Yaskawa INFORM job: new_kufsa_updated.JBI

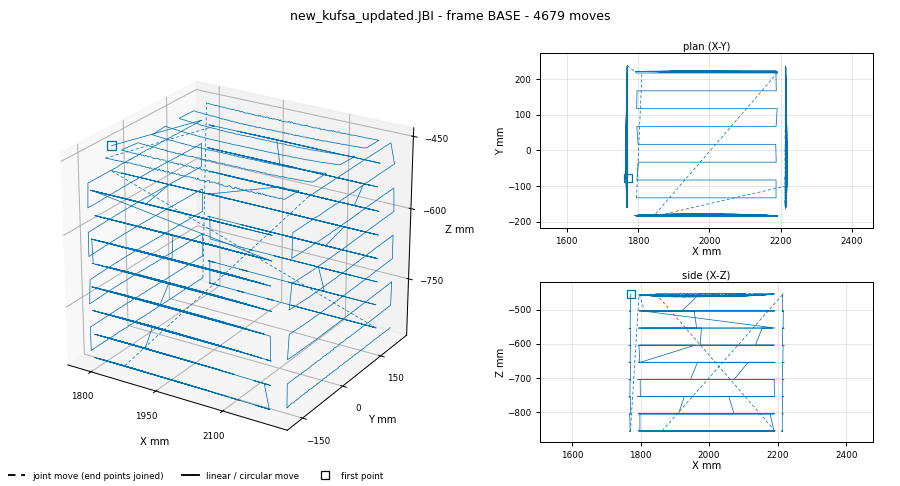
[picture p0: tool path of new_kufsa_updated.JBI in frame BASE, 4679 of 4679 moves have a stored position in this frame; points joined in program order, loops and branches not executed]
/JOB
//NAME NEW_KUFSA
//POS
///NPOS 4679,0,0,0,0,0
///TOOL 0
///POSTYPE BASE
///RECTAN
///RCONF 1,0,0,0,0,0,0,0,0,0,0,0,0,0,0,0,0,0,0,0,0,0,0,0
C00000=1771.695900,-78.143700,-454.553300,-91.472712,-88.665219,-178.527919
C00001=1770.552300,237.577800,-504.553300,-91.472712,-88.665219,-178.527919
C00002=1770.327900,234.301700,-504.553300,-91.472712,-88.665219,-178.527919
C00003=1770.357500,229.959000,-504.553300,-91.472712,-88.665219,-178.527919
C00004=1770.715100,226.685000,-504.553300,-91.472712,-88.665219,-178.527919
C00005=1770.694700,222.913600,-504.553300,-91.472712,-88.665219,-178.527919
C00006=1770.618200,221.900700,-504.553300,-91.472712,-88.665219,-178.527919
C00007=1770.622400,218.998600,-504.553300,-91.472712,-88.665219,-178.527919
C00008=1770.451600,217.707000,-504.553300,-91.472712,-88.665219,-178.527919
C00009=1770.752700,214.366400,-504.553300,-91.472712,-88.665219,-178.527919
C00010=1770.697000,210.035600,-504.553300,-91.472712,-88.665219,-178.527919
C00011=1770.753100,207.951700,-504.553300,-91.472712,-88.665219,-178.527919
C00012=1770.680200,203.374600,-504.553300,-91.472712,-88.665219,-178.527919
C00013=1770.529700,199.363700,-504.553300,-91.472712,-88.665219,-178.527919
C00014=1770.704300,193.088900,-504.553300,-91.472712,-88.665219,-178.527919
C00015=1770.481900,189.234700,-504.553300,-91.472712,-88.665219,-178.527919
C00016=1770.674300,186.293400,-504.553300,-91.472712,-88.665219,-178.527919
C00017=1770.533500,181.144000,-504.553300,-91.472712,-88.665219,-178.527919
C00018=1770.619900,177.321600,-504.553300,-91.472712,-88.665219,-178.527919
C00019=1770.311100,172.891400,-504.553300,-91.472712,-88.665219,-178.527919
C00020=1770.213900,166.678800,-504.553300,-91.472712,-88.665219,-178.527919
C00021=1770.097800,164.479000,-504.553300,-91.472712,-88.665219,-178.527919
C00022=1769.937500,159.949500,-504.553300,-91.472712,-88.665219,-178.527919
C00023=1770.653000,157.893100,-504.553300,-91.472712,-88.665219,-178.527919
C00024=1770.749700,154.381500,-504.553300,-91.472712,-88.665219,-178.527919
C00025=1770.288500,151.107400,-504.553300,-91.472712,-88.665219,-178.527919
C00026=1770.668700,148.632000,-504.553300,-91.472712,-88.665219,-178.527919
C00027=1770.398300,145.757600,-504.553300,-91.472712,-88.665219,-178.527919
C00028=1769.498100,142.997800,-504.553300,-91.472712,-88.665219,-178.527919
C00029=1769.363100,139.160700,-504.553300,-91.472712,-88.665219,-178.527919
C00030=1769.459100,135.555500,-504.553300,-91.472712,-88.665219,-178.527919
C00031=1769.040900,132.650400,-504.553300,-91.472712,-88.665219,-178.527919
C00032=1769.898800,130.507300,-504.553300,-91.472712,-88.665219,-178.527919
C00033=1770.728700,127.335900,-504.553300,-91.472712,-88.665219,-178.527919
C00034=1770.427200,123.559800,-504.553300,-91.472712,-88.665219,-178.527919
C00035=1768.954900,119.644000,-504.553300,-91.472712,-88.665219,-178.527919
C00036=1769.993600,117.378600,-504.553300,-91.472712,-88.665219,-178.527919
C00037=1768.828100,114.262100,-504.553300,-91.472712,-88.665219,-178.527919
C00038=1770.115200,111.383800,-504.553300,-91.472712,-88.665219,-178.527919
C00039=1769.668100,108.550000,-504.553300,-91.472712,-88.665219,-178.527919
C00040=1768.761100,104.884700,-504.553300,-91.472712,-88.665219,-178.527919
C00041=1769.568000,102.393100,-504.553300,-91.472712,-88.665219,-178.527919
C00042=1770.193300,98.407500,-504.553300,-91.472712,-88.665219,-178.527919
C00043=1768.903700,96.183100,-504.553300,-91.472712,-88.665219,-178.527919
C00044=1768.807500,91.494800,-504.553300,-91.472712,-88.665219,-178.527919
C00045=1769.610500,88.437300,-504.553300,-91.472712,-88.665219,-178.527919
C00046=1769.643300,85.334200,-504.553300,-91.472712,-88.665219,-178.527919
C00047=1770.204500,83.163200,-504.553300,-91.472712,-88.665219,-178.527919
C00048=1769.143800,79.495600,-504.553300,-91.472712,-88.665219,-178.527919
C00049=1770.143500,76.022500,-504.553300,-91.472712,-88.665219,-178.527919
C00050=1770.166100,73.523800,-504.553300,-91.472712,-88.665219,-178.527919
C00051=1768.794300,69.839900,-504.553300,-91.472712,-88.665219,-178.527919
C00052=1768.256500,65.364800,-504.553300,-91.472712,-88.665219,-178.527919
C00053=1769.079700,62.108500,-504.553300,-91.472712,-88.665219,-178.527919
C00054=1769.961500,58.974300,-504.553300,-91.472712,-88.665219,-178.527919
C00055=1770.647500,53.217300,-504.553300,-91.472712,-88.665219,-178.527919
C00056=1769.116700,51.163800,-504.553300,-91.472712,-88.665219,-178.527919
C00057=1768.800500,45.123900,-504.553300,-91.472712,-88.665219,-178.527919
C00058=1768.002400,42.027000,-504.553300,-91.472712,-88.665219,-178.527919
C00059=1768.569100,38.028400,-504.553300,-91.472712,-88.665219,-178.527919
C00060=1769.872300,32.986500,-504.553300,-91.472712,-88.665219,-178.527919
C00061=1768.268600,29.407100,-504.553300,-91.472712,-88.665219,-178.527919
C00062=1768.741300,27.721600,-504.553300,-91.472712,-88.665219,-178.527919
C00063=1768.516100,24.486500,-504.553300,-91.472712,-88.665219,-178.527919
C00064=1768.709900,22.063000,-504.553300,-91.472712,-88.665219,-178.527919
C00065=1770.169000,18.529100,-504.553300,-91.472712,-88.665219,-178.527919
C00066=1769.338300,14.603500,-504.553300,-91.472712,-88.665219,-178.527919
C00067=1769.785200,12.781600,-504.553300,-91.472712,-88.665219,-178.527919
C00068=1768.917400,10.596100,-504.553300,-91.472712,-88.665219,-178.527919
C00069=1770.959800,8.457400,-504.553300,-91.472712,-88.665219,-178.527919
C00070=1770.078300,4.762700,-504.553300,-91.472712,-88.665219,-178.527919
C00071=1770.056300,0.334200,-504.553300,-91.472712,-88.665219,-178.527919
C00072=1768.340800,-1.831400,-504.553300,-91.472712,-88.665219,-178.527919
C00073=1770.254300,-5.058200,-504.553300,-91.472712,-88.665219,-178.527919
C00074=1769.677500,-8.070100,-504.553300,-91.472712,-88.665219,-178.527919
C00075=1770.879300,-10.712700,-504.553300,-91.472712,-88.665219,-178.527919
C00076=1768.750700,-14.573600,-504.553300,-91.472712,-88.665219,-178.527919
C00077=1770.340400,-15.957100,-504.553300,-91.472712,-88.665219,-178.527919
C00078=1768.733600,-20.306900,-504.553300,-91.472712,-88.665219,-178.527919
C00079=1769.800500,-22.681600,-504.553300,-91.472712,-88.665219,-178.527919
C00080=1769.413100,-26.458000,-504.553300,-91.472712,-88.665219,-178.527919
C00081=1769.645800,-30.948700,-504.553300,-91.472712,-88.665219,-178.527919
C00082=1769.732900,-34.377100,-504.553300,-91.472712,-88.665219,-178.527919
C00083=1769.999900,-36.989700,-504.553300,-91.472712,-88.665219,-178.527919
C00084=1768.941700,-40.940500,-504.553300,-91.472712,-88.665219,-178.527919
C00085=1769.293400,-44.109800,-504.553300,-91.472712,-88.665219,-178.527919
C00086=1769.076200,-46.979100,-504.553300,-91.472712,-88.665219,-178.527919
C00087=1769.685800,-51.575500,-504.553300,-91.472712,-88.665219,-178.527919
C00088=1769.818600,-53.702900,-504.553300,-91.472712,-88.665219,-178.527919
C00089=1771.044100,-58.594600,-504.553300,-91.472712,-88.665219,-178.527919
C00090=1770.444400,-61.359500,-504.553300,-91.472712,-88.665219,-178.527919
C00091=1771.083300,-65.467700,-504.553300,-91.472712,-88.665219,-178.527919
C00092=1770.718600,-67.730300,-504.553300,-91.472712,-88.665219,-178.527919
C00093=1770.401400,-71.308800,-504.553300,-91.472712,-88.665219,-178.527919
C00094=1770.970400,-75.459300,-504.553300,-91.472712,-88.665219,-178.527919
C00095=1770.670500,-79.143800,-504.553300,-91.472712,-88.665219,-178.527919
C00096=1769.980400,-82.193500,-504.553300,-91.472712,-88.665219,-178.527919
C00097=1771.083500,-85.926000,-504.553300,-91.472712,-88.665219,-178.527919
C00098=1770.271700,-88.724100,-504.553300,-91.472712,-88.665219,-178.527919
C00099=1770.893900,-91.597400,-504.553300,-91.472712,-88.665219,-178.527919
C00100=1770.927400,-97.401600,-504.553300,-91.472712,-88.665219,-178.527919
C00101=1770.186700,-101.527400,-504.553300,-91.472712,-88.665219,-178.527919
C00102=1771.038900,-105.643300,-504.553300,-91.472712,-88.665219,-178.527919
C00103=1770.472200,-109.502300,-504.553300,-91.472712,-88.665219,-178.527919
C00104=1771.164000,-113.253700,-504.553300,-91.472712,-88.665219,-178.527919
C00105=1770.459300,-119.489700,-504.553300,-91.472712,-88.665219,-178.527919
C00106=1770.831500,-123.480600,-504.553300,-91.472712,-88.665219,-178.527919
C00107=1770.300700,-127.391200,-504.553300,-91.472712,-88.665219,-178.527919
C00108=1770.407700,-131.896000,-504.553300,-91.472712,-88.665219,-178.527919
C00109=1770.835300,-137.199200,-504.553300,-91.472712,-88.665219,-178.527919
C00110=1770.659300,-142.340600,-504.553300,-91.472712,-88.665219,-178.527919
C00111=1770.414300,-146.357400,-504.553300,-91.472712,-88.665219,-178.527919
C00112=1770.891300,-148.126700,-504.553300,-91.472712,-88.665219,-178.527919
C00113=1770.958700,-151.548700,-504.553300,-91.472712,-88.665219,-178.527919
C00114=1770.369300,-155.780700,-504.553300,-91.472712,-88.665219,-178.527919
C00115=1770.064400,-157.972700,-554.553300,-91.472712,-88.665219,-178.527919
C00116=1769.985800,-154.798600,-554.553300,-91.472712,-88.665219,-178.527919
C00117=1770.252900,-151.668100,-554.553300,-91.472712,-88.665219,-178.527919
C00118=1770.186000,-148.149800,-554.553300,-91.472712,-88.665219,-178.527919
C00119=1769.926300,-145.462600,-554.553300,-91.472712,-88.665219,-178.527919
C00120=1770.034700,-142.677400,-554.553300,-91.472712,-88.665219,-178.527919
C00121=1770.051100,-141.018200,-554.553300,-91.472712,-88.665219,-178.527919
C00122=1770.290900,-137.062400,-554.553300,-91.472712,-88.665219,-178.527919
C00123=1770.018000,-133.335900,-554.553300,-91.472712,-88.665219,-178.527919
C00124=1769.803300,-128.424000,-554.553300,-91.472712,-88.665219,-178.527919
C00125=1769.855600,-124.269200,-554.553300,-91.472712,-88.665219,-178.527919
C00126=1769.525500,-118.390000,-554.553300,-91.472712,-88.665219,-178.527919
C00127=1769.793500,-115.424000,-554.553300,-91.472712,-88.665219,-178.527919
C00128=1769.519200,-110.220900,-554.553300,-91.472712,-88.665219,-178.527919
C00129=1769.684400,-107.152900,-554.553300,-91.472712,-88.665219,-178.527919
C00130=1768.914900,-102.406800,-554.553300,-91.472712,-88.665219,-178.527919
C00131=1769.115300,-98.536800,-554.553300,-91.472712,-88.665219,-178.527919
C00132=1769.053600,-93.635300,-554.553300,-91.472712,-88.665219,-178.527919
C00133=1769.429700,-91.018400,-554.553300,-91.472712,-88.665219,-178.527919
C00134=1768.813100,-86.595600,-554.553300,-91.472712,-88.665219,-178.527919
C00135=1768.570100,-84.367200,-554.553300,-91.472712,-88.665219,-178.527919
C00136=1768.957000,-77.814700,-554.553300,-91.472712,-88.665219,-178.527919
C00137=1768.595600,-74.979800,-554.553300,-91.472712,-88.665219,-178.527919
C00138=1768.799500,-71.746300,-554.553300,-91.472712,-88.665219,-178.527919
C00139=1768.054600,-65.699200,-554.553300,-91.472712,-88.665219,-178.527919
C00140=1768.662200,-62.089600,-554.553300,-91.472712,-88.665219,-178.527919
C00141=1767.620000,-58.151700,-554.553300,-91.472712,-88.665219,-178.527919
C00142=1768.263100,-55.561800,-554.553300,-91.472712,-88.665219,-178.527919
C00143=1767.903700,-51.698200,-554.553300,-91.472712,-88.665219,-178.527919
C00144=1768.065400,-47.679100,-554.553300,-91.472712,-88.665219,-178.527919
C00145=1767.555200,-45.962900,-554.553300,-91.472712,-88.665219,-178.527919
C00146=1767.753200,-42.437500,-554.553300,-91.472712,-88.665219,-178.527919
C00147=1767.319200,-38.611400,-554.553300,-91.472712,-88.665219,-178.527919
C00148=1768.324800,-35.952800,-554.553300,-91.472712,-88.665219,-178.527919
C00149=1767.941400,-32.103400,-554.553300,-91.472712,-88.665219,-178.527919
C00150=1767.897400,-27.646600,-554.553300,-91.472712,-88.665219,-178.527919
C00151=1767.470100,-24.763700,-554.553300,-91.472712,-88.665219,-178.527919
C00152=1768.165500,-21.148800,-554.553300,-91.472712,-88.665219,-178.527919
C00153=1767.279600,-17.991700,-554.553300,-91.472712,-88.665219,-178.527919
C00154=1766.910000,-15.113500,-554.553300,-91.472712,-88.665219,-178.527919
C00155=1767.117100,-13.098900,-554.553300,-91.472712,-88.665219,-178.527919
C00156=1767.549600,-8.065000,-554.553300,-91.472712,-88.665219,-178.527919
C00157=1767.031300,-4.400700,-554.553300,-91.472712,-88.665219,-178.527919
C00158=1767.475000,-1.173300,-554.553300,-91.472712,-88.665219,-178.527919
C00159=1767.426600,2.602100,-554.553300,-91.472712,-88.665219,-178.527919
C00160=1767.176300,5.712400,-554.553300,-91.472712,-88.665219,-178.527919
C00161=1767.833000,9.832300,-554.553300,-91.472712,-88.665219,-178.527919
C00162=1766.890500,11.781500,-554.553300,-91.472712,-88.665219,-178.527919
C00163=1766.630100,14.852100,-554.553300,-91.472712,-88.665219,-178.527919
C00164=1766.855600,17.783900,-554.553300,-91.472712,-88.665219,-178.527919
C00165=1767.166900,23.127100,-554.553300,-91.472712,-88.665219,-178.527919
C00166=1766.808200,25.779000,-554.553300,-91.472712,-88.665219,-178.527919
C00167=1767.235900,29.472100,-554.553300,-91.472712,-88.665219,-178.527919
C00168=1767.482700,31.899300,-554.553300,-91.472712,-88.665219,-178.527919
C00169=1767.096100,36.646600,-554.553300,-91.472712,-88.665219,-178.527919
C00170=1767.341200,38.871800,-554.553300,-91.472712,-88.665219,-178.527919
C00171=1767.658000,43.665500,-554.553300,-91.472712,-88.665219,-178.527919
C00172=1767.751100,46.639000,-554.553300,-91.472712,-88.665219,-178.527919
C00173=1766.734900,49.320200,-554.553300,-91.472712,-88.665219,-178.527919
C00174=1767.010100,52.987400,-554.553300,-91.472712,-88.665219,-178.527919
C00175=1766.865400,54.632900,-554.553300,-91.472712,-88.665219,-178.527919
C00176=1766.975300,58.811400,-554.553300,-91.472712,-88.665219,-178.527919
C00177=1766.820100,62.675000,-554.553300,-91.472712,-88.665219,-178.527919
C00178=1767.473400,63.942300,-554.553300,-91.472712,-88.665219,-178.527919
C00179=1767.688000,69.184900,-554.553300,-91.472712,-88.665219,-178.527919
C00180=1767.663200,72.742000,-554.553300,-91.472712,-88.665219,-178.527919
C00181=1767.721400,74.587700,-554.553300,-91.472712,-88.665219,-178.527919
C00182=1767.129700,78.502200,-554.553300,-91.472712,-88.665219,-178.527919
C00183=1767.473300,82.128400,-554.553300,-91.472712,-88.665219,-178.527919
C00184=1767.850000,86.011900,-554.553300,-91.472712,-88.665219,-178.527919
C00185=1767.512700,88.481900,-554.553300,-91.472712,-88.665219,-178.527919
C00186=1767.498400,92.190800,-554.553300,-91.472712,-88.665219,-178.527919
C00187=1767.648900,95.142900,-554.553300,-91.472712,-88.665219,-178.527919
C00188=1768.013200,98.712800,-554.553300,-91.472712,-88.665219,-178.527919
C00189=1767.536000,102.630600,-554.553300,-91.472712,-88.665219,-178.527919
C00190=1768.341000,104.148200,-554.553300,-91.472712,-88.665219,-178.527919
C00191=1768.149100,109.466900,-554.553300,-91.472712,-88.665219,-178.527919
C00192=1767.809600,111.570700,-554.553300,-91.472712,-88.665219,-178.527919
C00193=1768.274600,115.042000,-554.553300,-91.472712,-88.665219,-178.527919
C00194=1768.051700,117.830100,-554.553300,-91.472712,-88.665219,-178.527919
C00195=1768.149400,121.772300,-554.553300,-91.472712,-88.665219,-178.527919
C00196=1768.267600,126.040600,-554.553300,-91.472712,-88.665219,-178.527919
C00197=1768.912100,129.892700,-554.553300,-91.472712,-88.665219,-178.527919
C00198=1768.578500,133.404000,-554.553300,-91.472712,-88.665219,-178.527919
C00199=1768.568000,137.189900,-554.553300,-91.472712,-88.665219,-178.527919
C00200=1768.626300,140.241600,-554.553300,-91.472712,-88.665219,-178.527919
C00201=1769.259200,144.757600,-554.553300,-91.472712,-88.665219,-178.527919
C00202=1769.491300,147.942200,-554.553300,-91.472712,-88.665219,-178.527919
C00203=1768.867800,152.469000,-554.553300,-91.472712,-88.665219,-178.527919
C00204=1769.033700,158.861000,-554.553300,-91.472712,-88.665219,-178.527919
C00205=1769.178000,162.098600,-554.553300,-91.472712,-88.665219,-178.527919
C00206=1769.440800,166.528800,-554.553300,-91.472712,-88.665219,-178.527919
C00207=1769.856300,170.531200,-554.553300,-91.472712,-88.665219,-178.527919
C00208=1769.542600,174.400200,-554.553300,-91.472712,-88.665219,-178.527919
C00209=1769.680300,178.042900,-554.553300,-91.472712,-88.665219,-178.527919
C00210=1769.645400,183.387600,-554.553300,-91.472712,-88.665219,-178.527919
C00211=1769.990800,186.124800,-554.553300,-91.472712,-88.665219,-178.527919
C00212=1769.966400,192.205400,-554.553300,-91.472712,-88.665219,-178.527919
C00213=1770.213500,197.858900,-554.553300,-91.472712,-88.665219,-178.527919
C00214=1770.368600,199.781300,-554.553300,-91.472712,-88.665219,-178.527919
C00215=1770.274200,204.121600,-554.553300,-91.472712,-88.665219,-178.527919
C00216=1770.392000,208.274700,-554.553300,-91.472712,-88.665219,-178.527919
C00217=1770.244600,211.666700,-554.553300,-91.472712,-88.665219,-178.527919
C00218=1770.348800,214.119800,-554.553300,-91.472712,-88.665219,-178.527919
C00219=1770.412900,216.228300,-554.553300,-91.472712,-88.665219,-178.527919
C00220=1770.288400,217.891800,-554.553300,-91.472712,-88.665219,-178.527919
C00221=1770.453300,221.090900,-554.553300,-91.472712,-88.665219,-178.527919
C00222=1770.352500,223.671700,-554.553300,-91.472712,-88.665219,-178.527919
C00223=1770.320200,226.845400,-554.553300,-91.472712,-88.665219,-178.527919
C00224=1770.293000,229.567500,-554.553300,-91.472712,-88.665219,-178.527919
C00225=1770.251200,232.163500,-554.553300,-91.472712,-88.665219,-178.527919
C00226=1770.287100,236.827400,-554.553300,-91.472712,-88.665219,-178.527919
C00227=1770.370200,235.106800,-604.553300,-91.472712,-88.665219,-178.527919
C00228=1770.306200,232.963000,-604.553300,-91.472712,-88.665219,-178.527919
C00229=1770.257600,228.166600,-604.553300,-91.472712,-88.665219,-178.527919
C00230=1770.450900,226.468100,-604.553300,-91.472712,-88.665219,-178.527919
C00231=1770.259500,223.189900,-604.553300,-91.472712,-88.665219,-178.527919
C00232=1770.277000,221.248000,-604.553300,-91.472712,-88.665219,-178.527919
C00233=1770.148500,218.427800,-604.553300,-91.472712,-88.665219,-178.527919
C00234=1770.194200,215.367100,-604.553300,-91.472712,-88.665219,-178.527919
C00235=1770.232000,212.866400,-604.553300,-91.472712,-88.665219,-178.527919
C00236=1770.171400,210.625400,-604.553300,-91.472712,-88.665219,-178.527919
C00237=1770.193000,208.326700,-604.553300,-91.472712,-88.665219,-178.527919
C00238=1770.192600,204.157000,-604.553300,-91.472712,-88.665219,-178.527919
C00239=1770.079300,201.309000,-604.553300,-91.472712,-88.665219,-178.527919
C00240=1769.910300,196.414300,-604.553300,-91.472712,-88.665219,-178.527919
C00241=1769.812400,190.026000,-604.553300,-91.472712,-88.665219,-178.527919
C00242=1769.792100,185.182300,-604.553300,-91.472712,-88.665219,-178.527919
C00243=1769.534600,181.326800,-604.553300,-91.472712,-88.665219,-178.527919
C00244=1769.432100,174.572200,-604.553300,-91.472712,-88.665219,-178.527919
C00245=1769.376300,171.854200,-604.553300,-91.472712,-88.665219,-178.527919
C00246=1769.273200,168.693300,-604.553300,-91.472712,-88.665219,-178.527919
C00247=1769.210100,164.632100,-604.553300,-91.472712,-88.665219,-178.527919
C00248=1769.225400,161.323900,-604.553300,-91.472712,-88.665219,-178.527919
C00249=1768.989400,157.131200,-604.553300,-91.472712,-88.665219,-178.527919
C00250=1768.884200,153.420700,-604.553300,-91.472712,-88.665219,-178.527919
C00251=1768.765700,149.271600,-604.553300,-91.472712,-88.665219,-178.527919
C00252=1768.560400,144.026200,-604.553300,-91.472712,-88.665219,-178.527919
C00253=1768.461400,142.475800,-604.553300,-91.472712,-88.665219,-178.527919
C00254=1768.416800,138.335800,-604.553300,-91.472712,-88.665219,-178.527919
C00255=1768.171400,135.000300,-604.553300,-91.472712,-88.665219,-178.527919
C00256=1768.070700,129.833300,-604.553300,-91.472712,-88.665219,-178.527919
C00257=1768.201000,128.249100,-604.553300,-91.472712,-88.665219,-178.527919
C00258=1768.024000,122.308800,-604.553300,-91.472712,-88.665219,-178.527919
C00259=1767.829500,118.132000,-604.553300,-91.472712,-88.665219,-178.527919
C00260=1767.814500,114.351100,-604.553300,-91.472712,-88.665219,-178.527919
C00261=1767.700500,111.498400,-604.553300,-91.472712,-88.665219,-178.527919
C00262=1767.456900,105.963100,-604.553300,-91.472712,-88.665219,-178.527919
C00263=1767.377100,103.365100,-604.553300,-91.472712,-88.665219,-178.527919
C00264=1767.384000,99.402100,-604.553300,-91.472712,-88.665219,-178.527919
C00265=1767.258900,95.013500,-604.553300,-91.472712,-88.665219,-178.527919
C00266=1767.308400,91.952600,-604.553300,-91.472712,-88.665219,-178.527919
C00267=1767.247400,87.764400,-604.553300,-91.472712,-88.665219,-178.527919
C00268=1767.149800,85.190600,-604.553300,-91.472712,-88.665219,-178.527919
C00269=1766.901700,81.256100,-604.553300,-91.472712,-88.665219,-178.527919
C00270=1766.933000,76.317800,-604.553300,-91.472712,-88.665219,-178.527919
C00271=1766.782800,74.446100,-604.553300,-91.472712,-88.665219,-178.527919
C00272=1766.859500,69.660800,-604.553300,-91.472712,-88.665219,-178.527919
C00273=1766.868200,66.185900,-604.553300,-91.472712,-88.665219,-178.527919
C00274=1766.661900,64.095500,-604.553300,-91.472712,-88.665219,-178.527919
C00275=1766.551400,58.727600,-604.553300,-91.472712,-88.665219,-178.527919
C00276=1766.729500,57.428200,-604.553300,-91.472712,-88.665219,-178.527919
C00277=1766.591400,53.805200,-604.553300,-91.472712,-88.665219,-178.527919
C00278=1766.492800,49.360000,-604.553300,-91.472712,-88.665219,-178.527919
C00279=1766.547900,47.714000,-604.553300,-91.472712,-88.665219,-178.527919
C00280=1766.651400,43.722700,-604.553300,-91.472712,-88.665219,-178.527919
C00281=1766.607500,41.117100,-604.553300,-91.472712,-88.665219,-178.527919
C00282=1766.590400,37.231400,-604.553300,-91.472712,-88.665219,-178.527919
C00283=1766.437600,33.936100,-604.553300,-91.472712,-88.665219,-178.527919
C00284=1766.385100,32.117300,-604.553300,-91.472712,-88.665219,-178.527919
C00285=1766.493300,28.329200,-604.553300,-91.472712,-88.665219,-178.527919
C00286=1766.379500,25.675700,-604.553300,-91.472712,-88.665219,-178.527919
C00287=1766.372600,21.756600,-604.553300,-91.472712,-88.665219,-178.527919
C00288=1766.514800,18.516500,-604.553300,-91.472712,-88.665219,-178.527919
C00289=1766.301500,13.809400,-604.553300,-91.472712,-88.665219,-178.527919
C00290=1766.484800,10.431400,-604.553300,-91.472712,-88.665219,-178.527919
C00291=1766.303200,7.858000,-604.553300,-91.472712,-88.665219,-178.527919
C00292=1766.405000,4.643600,-604.553300,-91.472712,-88.665219,-178.527919
C00293=1766.236300,0.530800,-604.553300,-91.472712,-88.665219,-178.527919
C00294=1766.370500,-1.758800,-604.553300,-91.472712,-88.665219,-178.527919
C00295=1766.620700,-6.784900,-604.553300,-91.472712,-88.665219,-178.527919
C00296=1766.551400,-10.765100,-604.553300,-91.472712,-88.665219,-178.527919
C00297=1766.359700,-18.133200,-604.553300,-91.472712,-88.665219,-178.527919
C00298=1766.561800,-22.644100,-604.553300,-91.472712,-88.665219,-178.527919
C00299=1766.482000,-28.365500,-604.553300,-91.472712,-88.665219,-178.527919
C00300=1766.858100,-33.249100,-604.553300,-91.472712,-88.665219,-178.527919
C00301=1766.585900,-37.166700,-604.553300,-91.472712,-88.665219,-178.527919
C00302=1766.650400,-39.795500,-604.553300,-91.472712,-88.665219,-178.527919
C00303=1766.829500,-45.406100,-604.553300,-91.472712,-88.665219,-178.527919
C00304=1766.919100,-48.696400,-604.553300,-91.472712,-88.665219,-178.527919
C00305=1767.456500,-53.356000,-604.553300,-91.472712,-88.665219,-178.527919
C00306=1767.039000,-57.576700,-604.553300,-91.472712,-88.665219,-178.527919
C00307=1766.838200,-61.993700,-604.553300,-91.472712,-88.665219,-178.527919
C00308=1767.415400,-65.020400,-604.553300,-91.472712,-88.665219,-178.527919
C00309=1767.107300,-69.137800,-604.553300,-91.472712,-88.665219,-178.527919
C00310=1767.288200,-71.447600,-604.553300,-91.472712,-88.665219,-178.527919
C00311=1767.775800,-76.946700,-604.553300,-91.472712,-88.665219,-178.527919
C00312=1767.689700,-77.718400,-604.553300,-91.472712,-88.665219,-178.527919
C00313=1767.565300,-82.097500,-604.553300,-91.472712,-88.665219,-178.527919
C00314=1768.141600,-85.962700,-604.553300,-91.472712,-88.665219,-178.527919
C00315=1767.609700,-90.076800,-604.553300,-91.472712,-88.665219,-178.527919
C00316=1767.737500,-92.140200,-604.553300,-91.472712,-88.665219,-178.527919
C00317=1768.117000,-98.215200,-604.553300,-91.472712,-88.665219,-178.527919
C00318=1768.411900,-101.146000,-604.553300,-91.472712,-88.665219,-178.527919
C00319=1768.629000,-106.026500,-604.553300,-91.472712,-88.665219,-178.527919
C00320=1768.512600,-110.209400,-604.553300,-91.472712,-88.665219,-178.527919
C00321=1768.575700,-114.402400,-604.553300,-91.472712,-88.665219,-178.527919
C00322=1768.873400,-119.976200,-604.553300,-91.472712,-88.665219,-178.527919
C00323=1768.893900,-124.081700,-604.553300,-91.472712,-88.665219,-178.527919
C00324=1769.200700,-127.094900,-604.553300,-91.472712,-88.665219,-178.527919
C00325=1769.326800,-130.861900,-604.553300,-91.472712,-88.665219,-178.527919
C00326=1769.431700,-135.482600,-604.553300,-91.472712,-88.665219,-178.527919
C00327=1769.605000,-138.245900,-604.553300,-91.472712,-88.665219,-178.527919
C00328=1769.602500,-140.883800,-604.553300,-91.472712,-88.665219,-178.527919
C00329=1769.564500,-142.714600,-604.553300,-91.472712,-88.665219,-178.527919
C00330=1769.767000,-145.788300,-604.553300,-91.472712,-88.665219,-178.527919
C00331=1769.875100,-150.321500,-604.553300,-91.472712,-88.665219,-178.527919
C00332=1769.940300,-152.355700,-604.553300,-91.472712,-88.665219,-178.527919
C00333=1769.978600,-154.348600,-604.553300,-91.472712,-88.665219,-178.527919
C00334=1770.081600,-156.453500,-604.553300,-91.472712,-88.665219,-178.527919
C00335=1770.509100,-159.529500,-604.553300,-91.472712,-88.665219,-178.527919
C00336=1770.117300,-159.575400,-654.553300,-91.472712,-88.665219,-178.527919
C00337=1770.320100,-156.526900,-654.553300,-91.472712,-88.665219,-178.527919
C00338=1770.123600,-154.839500,-654.553300,-91.472712,-88.665219,-178.527919
C00339=1769.867100,-151.664100,-654.553300,-91.472712,-88.665219,-178.527919
C00340=1769.884200,-148.439400,-654.553300,-91.472712,-88.665219,-178.527919
C00341=1769.553700,-145.816000,-654.553300,-91.472712,-88.665219,-178.527919
C00342=1769.374200,-141.011100,-654.553300,-91.472712,-88.665219,-178.527919
C00343=1769.382300,-137.357700,-654.553300,-91.472712,-88.665219,-178.527919
C00344=1769.263700,-133.039300,-654.553300,-91.472712,-88.665219,-178.527919
C00345=1769.137600,-128.576700,-654.553300,-91.472712,-88.665219,-178.527919
C00346=1768.717600,-124.502600,-654.553300,-91.472712,-88.665219,-178.527919
C00347=1768.670500,-119.952500,-654.553300,-91.472712,-88.665219,-178.527919
C00348=1768.524500,-116.185900,-654.553300,-91.472712,-88.665219,-178.527919
C00349=1768.277000,-110.809400,-654.553300,-91.472712,-88.665219,-178.527919
C00350=1767.976200,-108.437400,-654.553300,-91.472712,-88.665219,-178.527919
C00351=1767.996800,-104.560600,-654.553300,-91.472712,-88.665219,-178.527919
C00352=1767.911000,-100.961900,-654.553300,-91.472712,-88.665219,-178.527919
C00353=1767.587900,-96.903300,-654.553300,-91.472712,-88.665219,-178.527919
C00354=1767.627200,-91.101400,-654.553300,-91.472712,-88.665219,-178.527919
C00355=1767.596700,-86.525700,-654.553300,-91.472712,-88.665219,-178.527919
C00356=1767.486900,-83.250600,-654.553300,-91.472712,-88.665219,-178.527919
C00357=1767.203800,-78.389700,-654.553300,-91.472712,-88.665219,-178.527919
C00358=1767.125800,-74.980500,-654.553300,-91.472712,-88.665219,-178.527919
C00359=1766.983600,-70.081400,-654.553300,-91.472712,-88.665219,-178.527919
C00360=1766.915900,-65.925200,-654.553300,-91.472712,-88.665219,-178.527919
C00361=1766.667400,-62.605500,-654.553300,-91.472712,-88.665219,-178.527919
C00362=1766.744500,-59.713900,-654.553300,-91.472712,-88.665219,-178.527919
C00363=1766.653100,-55.722200,-654.553300,-91.472712,-88.665219,-178.527919
C00364=1766.723200,-52.201200,-654.553300,-91.472712,-88.665219,-178.527919
C00365=1766.718700,-48.654200,-654.553300,-91.472712,-88.665219,-178.527919
C00366=1766.590100,-46.788600,-654.553300,-91.472712,-88.665219,-178.527919
C00367=1766.515100,-42.707400,-654.553300,-91.472712,-88.665219,-178.527919
C00368=1766.359700,-40.226300,-654.553300,-91.472712,-88.665219,-178.527919
C00369=1766.323400,-35.374800,-654.553300,-91.472712,-88.665219,-178.527919
C00370=1766.411600,-33.040300,-654.553300,-91.472712,-88.665219,-178.527919
C00371=1766.306700,-29.523300,-654.553300,-91.472712,-88.665219,-178.527919
C00372=1766.341900,-26.435700,-654.553300,-91.472712,-88.665219,-178.527919
C00373=1766.173200,-23.157900,-654.553300,-91.472712,-88.665219,-178.527919
C00374=1766.177700,-19.788900,-654.553300,-91.472712,-88.665219,-178.527919
C00375=1766.332500,-17.216900,-654.553300,-91.472712,-88.665219,-178.527919
C00376=1766.202800,-11.560700,-654.553300,-91.472712,-88.665219,-178.527919
C00377=1766.227200,-6.814600,-654.553300,-91.472712,-88.665219,-178.527919
C00378=1766.301100,-4.236900,-654.553300,-91.472712,-88.665219,-178.527919
C00379=1766.194500,-2.309100,-654.553300,-91.472712,-88.665219,-178.527919
C00380=1766.308400,1.745700,-654.553300,-91.472712,-88.665219,-178.527919
C00381=1766.196900,4.838400,-654.553300,-91.472712,-88.665219,-178.527919
C00382=1766.376600,8.733200,-654.553300,-91.472712,-88.665219,-178.527919
C00383=1766.377100,13.039300,-654.553300,-91.472712,-88.665219,-178.527919
C00384=1766.438600,17.722700,-654.553300,-91.472712,-88.665219,-178.527919
C00385=1766.659100,21.967700,-654.553300,-91.472712,-88.665219,-178.527919
C00386=1766.403900,24.434500,-654.553300,-91.472712,-88.665219,-178.527919
C00387=1766.525600,28.527400,-654.553300,-91.472712,-88.665219,-178.527919
C00388=1766.503600,32.024800,-654.553300,-91.472712,-88.665219,-178.527919
C00389=1766.442600,35.647900,-654.553300,-91.472712,-88.665219,-178.527919
C00390=1766.502200,38.705400,-654.553300,-91.472712,-88.665219,-178.527919
C00391=1766.461800,42.432000,-654.553300,-91.472712,-88.665219,-178.527919
C00392=1766.825700,44.691200,-654.553300,-91.472712,-88.665219,-178.527919
C00393=1766.628400,48.336600,-654.553300,-91.472712,-88.665219,-178.527919
C00394=1766.623900,52.387400,-654.553300,-91.472712,-88.665219,-178.527919
C00395=1766.758400,56.149600,-654.553300,-91.472712,-88.665219,-178.527919
C00396=1766.882100,60.694900,-654.553300,-91.472712,-88.665219,-178.527919
C00397=1766.925000,63.398900,-654.553300,-91.472712,-88.665219,-178.527919
C00398=1766.767500,68.222900,-654.553300,-91.472712,-88.665219,-178.527919
C00399=1766.823900,71.359400,-654.553300,-91.472712,-88.665219,-178.527919
C00400=1767.340100,73.808600,-654.553300,-91.472712,-88.665219,-178.527919
C00401=1767.108300,78.216400,-654.553300,-91.472712,-88.665219,-178.527919
C00402=1767.216700,81.040500,-654.553300,-91.472712,-88.665219,-178.527919
C00403=1767.053300,83.598700,-654.553300,-91.472712,-88.665219,-178.527919
C00404=1767.389300,86.886600,-654.553300,-91.472712,-88.665219,-178.527919
C00405=1767.325500,89.075500,-654.553300,-91.472712,-88.665219,-178.527919
C00406=1767.328100,93.768200,-654.553300,-91.472712,-88.665219,-178.527919
C00407=1767.375300,97.880100,-654.553300,-91.472712,-88.665219,-178.527919
C00408=1767.615100,99.876100,-654.553300,-91.472712,-88.665219,-178.527919
C00409=1767.609900,103.163000,-654.553300,-91.472712,-88.665219,-178.527919
C00410=1767.887300,107.865500,-654.553300,-91.472712,-88.665219,-178.527919
C00411=1767.665000,110.542900,-654.553300,-91.472712,-88.665219,-178.527919
C00412=1767.940300,114.339800,-654.553300,-91.472712,-88.665219,-178.527919
C00413=1767.898100,117.119500,-654.553300,-91.472712,-88.665219,-178.527919
C00414=1768.088500,120.361800,-654.553300,-91.472712,-88.665219,-178.527919
C00415=1768.236200,123.715900,-654.553300,-91.472712,-88.665219,-178.527919
C00416=1768.394100,128.171700,-654.553300,-91.472712,-88.665219,-178.527919
C00417=1768.429000,132.477900,-654.553300,-91.472712,-88.665219,-178.527919
C00418=1768.595900,136.278700,-654.553300,-91.472712,-88.665219,-178.527919
C00419=1768.509100,138.597000,-654.553300,-91.472712,-88.665219,-178.527919
C00420=1768.744800,143.279900,-654.553300,-91.472712,-88.665219,-178.527919
C00421=1768.552700,145.422200,-654.553300,-91.472712,-88.665219,-178.527919
C00422=1768.813800,150.793200,-654.553300,-91.472712,-88.665219,-178.527919
C00423=1768.949400,153.570700,-654.553300,-91.472712,-88.665219,-178.527919
C00424=1769.099600,158.112300,-654.553300,-91.472712,-88.665219,-178.527919
C00425=1769.193300,162.332700,-654.553300,-91.472712,-88.665219,-178.527919
C00426=1769.148400,164.490500,-654.553300,-91.472712,-88.665219,-178.527919
C00427=1769.480200,169.180500,-654.553300,-91.472712,-88.665219,-178.527919
C00428=1769.415000,172.758600,-654.553300,-91.472712,-88.665219,-178.527919
C00429=1769.626900,176.485800,-654.553300,-91.472712,-88.665219,-178.527919
C00430=1769.532500,179.329400,-654.553300,-91.472712,-88.665219,-178.527919
C00431=1769.624500,182.919000,-654.553300,-91.472712,-88.665219,-178.527919
C00432=1769.613300,185.571500,-654.553300,-91.472712,-88.665219,-178.527919
C00433=1769.719400,188.426000,-654.553300,-91.472712,-88.665219,-178.527919
C00434=1769.836900,192.754400,-654.553300,-91.472712,-88.665219,-178.527919
C00435=1769.825300,196.480500,-654.553300,-91.472712,-88.665219,-178.527919
C00436=1769.938900,198.390700,-654.553300,-91.472712,-88.665219,-178.527919
C00437=1769.994300,201.167800,-654.553300,-91.472712,-88.665219,-178.527919
C00438=1769.906800,204.468200,-654.553300,-91.472712,-88.665219,-178.527919
C00439=1770.035400,208.734900,-654.553300,-91.472712,-88.665219,-178.527919
C00440=1770.211900,211.790700,-654.553300,-91.472712,-88.665219,-178.527919
C00441=1770.231300,214.977900,-654.553300,-91.472712,-88.665219,-178.527919
C00442=1770.210800,217.834100,-654.553300,-91.472712,-88.665219,-178.527919
C00443=1770.051800,220.537800,-654.553300,-91.472712,-88.665219,-178.527919
C00444=1770.262700,224.162300,-654.553300,-91.472712,-88.665219,-178.527919
C00445=1770.243900,227.332900,-654.553300,-91.472712,-88.665219,-178.527919
C00446=1770.266200,229.425200,-654.553300,-91.472712,-88.665219,-178.527919
C00447=1770.197200,232.271600,-654.553300,-91.472712,-88.665219,-178.527919
C00448=1770.214900,234.047600,-654.553300,-91.472712,-88.665219,-178.527919
C00449=1770.367600,236.678800,-654.553300,-91.472712,-88.665219,-178.527919
C00450=1770.629700,237.886900,-654.553300,-91.472712,-88.665219,-178.527919
C00451=1770.809500,237.783500,-704.553300,-91.472712,-88.665219,-178.527919
C00452=1770.202400,233.462500,-704.553300,-91.472712,-88.665219,-178.527919
C00453=1770.185800,232.561300,-704.553300,-91.472712,-88.665219,-178.527919
C00454=1770.350200,229.876200,-704.553300,-91.472712,-88.665219,-178.527919
C00455=1770.399000,227.105200,-704.553300,-91.472712,-88.665219,-178.527919
C00456=1770.340100,223.999100,-704.553300,-91.472712,-88.665219,-178.527919
C00457=1770.128100,218.795600,-704.553300,-91.472712,-88.665219,-178.527919
C00458=1770.130900,214.749500,-704.553300,-91.472712,-88.665219,-178.527919
C00459=1770.138100,212.755900,-704.553300,-91.472712,-88.665219,-178.527919
C00460=1770.150800,208.342600,-704.553300,-91.472712,-88.665219,-178.527919
C00461=1770.104100,206.513500,-704.553300,-91.472712,-88.665219,-178.527919
C00462=1769.870900,201.721200,-704.553300,-91.472712,-88.665219,-178.527919
C00463=1769.743700,197.610900,-704.553300,-91.472712,-88.665219,-178.527919
C00464=1769.775100,194.054800,-704.553300,-91.472712,-88.665219,-178.527919
C00465=1769.672900,190.083700,-704.553300,-91.472712,-88.665219,-178.527919
C00466=1769.702200,185.565400,-704.553300,-91.472712,-88.665219,-178.527919
C00467=1769.612600,182.727500,-704.553300,-91.472712,-88.665219,-178.527919
C00468=1769.460700,179.381800,-704.553300,-91.472712,-88.665219,-178.527919
C00469=1769.648900,176.724300,-704.553300,-91.472712,-88.665219,-178.527919
C00470=1769.340400,171.289700,-704.553300,-91.472712,-88.665219,-178.527919
C00471=1769.267900,167.789300,-704.553300,-91.472712,-88.665219,-178.527919
C00472=1769.175600,164.192900,-704.553300,-91.472712,-88.665219,-178.527919
C00473=1769.444300,159.869800,-704.553300,-91.472712,-88.665219,-178.527919
C00474=1769.263400,156.296100,-704.553300,-91.472712,-88.665219,-178.527919
C00475=1769.147300,152.726400,-704.553300,-91.472712,-88.665219,-178.527919
C00476=1769.003700,149.613500,-704.553300,-91.472712,-88.665219,-178.527919
C00477=1768.789400,147.505000,-704.553300,-91.472712,-88.665219,-178.527919
C00478=1768.991200,144.214700,-704.553300,-91.472712,-88.665219,-178.527919
C00479=1768.643300,139.590300,-704.553300,-91.472712,-88.665219,-178.527919
C00480=1768.551700,138.826700,-704.553300,-91.472712,-88.665219,-178.527919
C00481=1768.903000,133.695200,-704.553300,-91.472712,-88.665219,-178.527919
C00482=1768.577100,131.492400,-704.553300,-91.472712,-88.665219,-178.527919
C00483=1768.331700,127.558200,-704.553300,-91.472712,-88.665219,-178.527919
C00484=1768.377400,123.910500,-704.553300,-91.472712,-88.665219,-178.527919
C00485=1768.376300,121.085100,-704.553300,-91.472712,-88.665219,-178.527919
C00486=1768.380200,116.784600,-704.553300,-91.472712,-88.665219,-178.527919
C00487=1768.163700,113.608900,-704.553300,-91.472712,-88.665219,-178.527919
C00488=1768.115300,107.819200,-704.553300,-91.472712,-88.665219,-178.527919
C00489=1767.917700,105.570200,-704.553300,-91.472712,-88.665219,-178.527919
C00490=1768.170000,101.793400,-704.553300,-91.472712,-88.665219,-178.527919
C00491=1768.025400,96.957500,-704.553300,-91.472712,-88.665219,-178.527919
C00492=1767.799500,93.547600,-704.553300,-91.472712,-88.665219,-178.527919
C00493=1768.063000,89.858300,-704.553300,-91.472712,-88.665219,-178.527919
C00494=1768.099600,88.013300,-704.553300,-91.472712,-88.665219,-178.527919
C00495=1768.060200,83.837200,-704.553300,-91.472712,-88.665219,-178.527919
C00496=1767.560100,79.867200,-704.553300,-91.472712,-88.665219,-178.527919
C00497=1767.679300,74.754900,-704.553300,-91.472712,-88.665219,-178.527919
C00498=1767.808900,72.903200,-704.553300,-91.472712,-88.665219,-178.527919
C00499=1767.316100,68.310200,-704.553300,-91.472712,-88.665219,-178.527919
C00500=1767.747600,65.275200,-704.553300,-91.472712,-88.665219,-178.527919
C00501=1767.201400,61.788200,-704.553300,-91.472712,-88.665219,-178.527919
C00502=1767.403400,59.188900,-704.553300,-91.472712,-88.665219,-178.527919
C00503=1767.092000,55.798300,-704.553300,-91.472712,-88.665219,-178.527919
C00504=1767.384700,49.885900,-704.553300,-91.472712,-88.665219,-178.527919
C00505=1767.487200,47.500200,-704.553300,-91.472712,-88.665219,-178.527919
C00506=1766.843100,42.985200,-704.553300,-91.472712,-88.665219,-178.527919
C00507=1767.188700,37.478500,-704.553300,-91.472712,-88.665219,-178.527919
C00508=1767.164100,35.068000,-704.553300,-91.472712,-88.665219,-178.527919
C00509=1766.544400,28.667600,-704.553300,-91.472712,-88.665219,-178.527919
C00510=1766.513700,23.003000,-704.553300,-91.472712,-88.665219,-178.527919
C00511=1766.707900,18.097800,-704.553300,-91.472712,-88.665219,-178.527919
C00512=1766.988100,13.654700,-704.553300,-91.472712,-88.665219,-178.527919
C00513=1766.658000,9.177200,-704.553300,-91.472712,-88.665219,-178.527919
C00514=1766.434600,5.103600,-704.553300,-91.472712,-88.665219,-178.527919
C00515=1766.518600,0.670300,-704.553300,-91.472712,-88.665219,-178.527919
C00516=1766.415100,-4.379100,-704.553300,-91.472712,-88.665219,-178.527919
C00517=1766.573000,-6.413900,-704.553300,-91.472712,-88.665219,-178.527919
C00518=1766.545800,-10.605300,-704.553300,-91.472712,-88.665219,-178.527919
C00519=1766.356200,-12.346500,-704.553300,-91.472712,-88.665219,-178.527919
C00520=1766.561500,-17.796700,-704.553300,-91.472712,-88.665219,-178.527919
C00521=1766.327900,-20.384200,-704.553300,-91.472712,-88.665219,-178.527919
C00522=1766.123000,-22.691700,-704.553300,-91.472712,-88.665219,-178.527919
C00523=1766.194100,-25.522900,-704.553300,-91.472712,-88.665219,-178.527919
C00524=1766.322000,-30.586200,-704.553300,-91.472712,-88.665219,-178.527919
C00525=1766.318200,-32.979500,-704.553300,-91.472712,-88.665219,-178.527919
C00526=1766.313700,-38.033300,-704.553300,-91.472712,-88.665219,-178.527919
C00527=1766.288900,-42.511100,-704.553300,-91.472712,-88.665219,-178.527919
C00528=1766.352700,-45.291900,-704.553300,-91.472712,-88.665219,-178.527919
C00529=1766.325500,-49.238000,-704.553300,-91.472712,-88.665219,-178.527919
C00530=1766.421400,-53.006000,-704.553300,-91.472712,-88.665219,-178.527919
C00531=1766.496300,-54.554000,-704.553300,-91.472712,-88.665219,-178.527919
C00532=1766.516900,-60.754100,-704.553300,-91.472712,-88.665219,-178.527919
C00533=1766.509200,-65.176500,-704.553300,-91.472712,-88.665219,-178.527919
C00534=1766.556900,-67.018500,-704.553300,-91.472712,-88.665219,-178.527919
C00535=1766.732300,-72.363200,-704.553300,-91.472712,-88.665219,-178.527919
C00536=1766.799500,-75.660900,-704.553300,-91.472712,-88.665219,-178.527919
C00537=1766.732600,-77.517000,-704.553300,-91.472712,-88.665219,-178.527919
C00538=1766.843100,-81.232700,-704.553300,-91.472712,-88.665219,-178.527919
C00539=1766.752100,-84.928700,-704.553300,-91.472712,-88.665219,-178.527919
C00540=1766.888400,-90.510200,-704.553300,-91.472712,-88.665219,-178.527919
C00541=1767.104900,-97.060700,-704.553300,-91.472712,-88.665219,-178.527919
C00542=1767.375700,-103.159200,-704.553300,-91.472712,-88.665219,-178.527919
C00543=1767.774800,-110.456300,-704.553300,-91.472712,-88.665219,-178.527919
C00544=1767.773700,-113.285800,-704.553300,-91.472712,-88.665219,-178.527919
C00545=1767.830500,-117.876800,-704.553300,-91.472712,-88.665219,-178.527919
C00546=1768.001500,-121.289400,-704.553300,-91.472712,-88.665219,-178.527919
C00547=1768.342200,-126.108700,-704.553300,-91.472712,-88.665219,-178.527919
C00548=1768.356700,-132.014300,-704.553300,-91.472712,-88.665219,-178.527919
C00549=1768.610600,-134.691700,-704.553300,-91.472712,-88.665219,-178.527919
C00550=1768.762500,-138.493500,-704.553300,-91.472712,-88.665219,-178.527919
C00551=1768.788000,-142.674300,-704.553300,-91.472712,-88.665219,-178.527919
C00552=1768.959500,-147.358900,-704.553300,-91.472712,-88.665219,-178.527919
C00553=1769.295500,-152.510700,-704.553300,-91.472712,-88.665219,-178.527919
C00554=1769.744700,-155.525800,-704.553300,-91.472712,-88.665219,-178.527919
C00555=1769.677800,-157.446700,-704.553300,-91.472712,-88.665219,-178.527919
C00556=1769.177300,-160.393000,-754.553300,-91.472712,-88.665219,-178.527919
C00557=1769.016600,-156.123300,-754.553300,-91.472712,-88.665219,-178.527919
C00558=1769.042400,-152.132700,-754.553300,-91.472712,-88.665219,-178.527919
C00559=1769.089900,-151.156300,-754.553300,-91.472712,-88.665219,-178.527919
C00560=1768.846900,-147.562000,-754.553300,-91.472712,-88.665219,-178.527919
C00561=1768.760800,-143.668600,-754.553300,-91.472712,-88.665219,-178.527919
C00562=1768.739200,-140.362500,-754.553300,-91.472712,-88.665219,-178.527919
C00563=1768.551700,-137.707000,-754.553300,-91.472712,-88.665219,-178.527919
C00564=1768.247700,-132.131200,-754.553300,-91.472712,-88.665219,-178.527919
C00565=1768.111500,-127.689200,-754.553300,-91.472712,-88.665219,-178.527919
C00566=1768.117000,-122.626700,-754.553300,-91.472712,-88.665219,-178.527919
C00567=1768.055700,-116.298400,-754.553300,-91.472712,-88.665219,-178.527919
C00568=1767.622400,-111.601300,-754.553300,-91.472712,-88.665219,-178.527919
C00569=1767.587900,-108.986400,-754.553300,-91.472712,-88.665219,-178.527919
C00570=1767.281200,-104.592700,-754.553300,-91.472712,-88.665219,-178.527919
C00571=1767.413300,-101.088500,-754.553300,-91.472712,-88.665219,-178.527919
C00572=1767.384400,-97.494900,-754.553300,-91.472712,-88.665219,-178.527919
C00573=1767.082200,-91.991000,-754.553300,-91.472712,-88.665219,-178.527919
C00574=1767.291000,-89.016300,-754.553300,-91.472712,-88.665219,-178.527919
C00575=1767.085300,-86.564500,-754.553300,-91.472712,-88.665219,-178.527919
C00576=1767.122600,-81.689100,-754.553300,-91.472712,-88.665219,-178.527919
C00577=1767.321700,-79.629900,-754.553300,-91.472712,-88.665219,-178.527919
C00578=1766.973100,-74.033800,-754.553300,-91.472712,-88.665219,-178.527919
C00579=1766.831100,-71.964900,-754.553300,-91.472712,-88.665219,-178.527919
C00580=1766.932000,-68.088400,-754.553300,-91.472712,-88.665219,-178.527919
C00581=1767.060900,-65.001900,-754.553300,-91.472712,-88.665219,-178.527919
C00582=1766.766800,-60.738200,-754.553300,-91.472712,-88.665219,-178.527919
C00583=1766.513000,-56.938800,-754.553300,-91.472712,-88.665219,-178.527919
C00584=1766.666400,-53.552300,-754.553300,-91.472712,-88.665219,-178.527919
C00585=1766.623900,-50.572100,-754.553300,-91.472712,-88.665219,-178.527919
C00586=1767.080800,-44.421000,-754.553300,-91.472712,-88.665219,-178.527919
C00587=1767.011800,-40.596200,-754.553300,-91.472712,-88.665219,-178.527919
C00588=1767.004100,-35.459900,-754.553300,-91.472712,-88.665219,-178.527919
C00589=1766.828100,-32.298900,-754.553300,-91.472712,-88.665219,-178.527919
C00590=1767.177000,-28.049900,-754.553300,-91.472712,-88.665219,-178.527919
C00591=1766.962300,-23.962300,-754.553300,-91.472712,-88.665219,-178.527919
C00592=1767.034100,-20.172400,-754.553300,-91.472712,-88.665219,-178.527919
C00593=1767.064400,-16.256100,-754.553300,-91.472712,-88.665219,-178.527919
C00594=1766.895000,-10.834000,-754.553300,-91.472712,-88.665219,-178.527919
C00595=1767.108700,-5.982500,-754.553300,-91.472712,-88.665219,-178.527919
C00596=1767.041800,-3.001700,-754.553300,-91.472712,-88.665219,-178.527919
C00597=1767.429000,0.596000,-754.553300,-91.472712,-88.665219,-178.527919
C00598=1767.136200,3.876500,-754.553300,-91.472712,-88.665219,-178.527919
C00599=1767.213100,8.277900,-754.553300,-91.472712,-88.665219,-178.527919
C00600=1766.987000,12.321300,-754.553300,-91.472712,-88.665219,-178.527919
C00601=1767.034800,17.330600,-754.553300,-91.472712,-88.665219,-178.527919
C00602=1767.507100,18.423900,-754.553300,-91.472712,-88.665219,-178.527919
C00603=1767.701200,22.699800,-754.553300,-91.472712,-88.665219,-178.527919
C00604=1767.453700,25.670600,-754.553300,-91.472712,-88.665219,-178.527919
C00605=1767.691100,28.869900,-754.553300,-91.472712,-88.665219,-178.527919
C00606=1768.141800,33.114300,-754.553300,-91.472712,-88.665219,-178.527919
C00607=1767.743000,38.747700,-754.553300,-91.472712,-88.665219,-178.527919
C00608=1767.666700,41.228900,-754.553300,-91.472712,-88.665219,-178.527919
C00609=1767.526900,45.615200,-754.553300,-91.472712,-88.665219,-178.527919
C00610=1767.840500,48.545500,-754.553300,-91.472712,-88.665219,-178.527919
C00611=1767.862100,52.517700,-754.553300,-91.472712,-88.665219,-178.527919
C00612=1768.495900,55.753100,-754.553300,-91.472712,-88.665219,-178.527919
C00613=1768.536000,59.911100,-754.553300,-91.472712,-88.665219,-178.527919
C00614=1768.416100,65.997800,-754.553300,-91.472712,-88.665219,-178.527919
C00615=1768.502200,68.312400,-754.553300,-91.472712,-88.665219,-178.527919
C00616=1768.597000,73.780900,-754.553300,-91.472712,-88.665219,-178.527919
C00617=1768.475700,74.990100,-754.553300,-91.472712,-88.665219,-178.527919
C00618=1768.144200,79.819900,-754.553300,-91.472712,-88.665219,-178.527919
C00619=1768.645400,82.344300,-754.553300,-91.472712,-88.665219,-178.527919
C00620=1768.563500,86.086600,-754.553300,-91.472712,-88.665219,-178.527919
C00621=1768.707800,90.720200,-754.553300,-91.472712,-88.665219,-178.527919
C00622=1768.273500,94.737200,-754.553300,-91.472712,-88.665219,-178.527919
C00623=1768.473200,98.255100,-754.553300,-91.472712,-88.665219,-178.527919
C00624=1768.812700,99.932900,-754.553300,-91.472712,-88.665219,-178.527919
C00625=1768.544700,104.431000,-754.553300,-91.472712,-88.665219,-178.527919
C00626=1768.604000,106.974600,-754.553300,-91.472712,-88.665219,-178.527919
C00627=1768.582300,111.148000,-754.553300,-91.472712,-88.665219,-178.527919
C00628=1769.022600,113.408200,-754.553300,-91.472712,-88.665219,-178.527919
C00629=1768.793900,119.081300,-754.553300,-91.472712,-88.665219,-178.527919
C00630=1769.076900,122.732400,-754.553300,-91.472712,-88.665219,-178.527919
C00631=1768.802400,128.517400,-754.553300,-91.472712,-88.665219,-178.527919
C00632=1769.365900,130.063000,-754.553300,-91.472712,-88.665219,-178.527919
C00633=1769.009700,134.510400,-754.553300,-91.472712,-88.665219,-178.527919
C00634=1768.983900,139.175100,-754.553300,-91.472712,-88.665219,-178.527919
C00635=1769.441200,142.838700,-754.553300,-91.472712,-88.665219,-178.527919
C00636=1769.260600,147.369500,-754.553300,-91.472712,-88.665219,-178.527919
C00637=1769.539800,150.143600,-754.553300,-91.472712,-88.665219,-178.527919
C00638=1769.572900,154.878100,-754.553300,-91.472712,-88.665219,-178.527919
C00639=1769.488800,157.934100,-754.553300,-91.472712,-88.665219,-178.527919
C00640=1769.462800,161.968200,-754.553300,-91.472712,-88.665219,-178.527919
C00641=1769.586500,165.848700,-754.553300,-91.472712,-88.665219,-178.527919
C00642=1769.722400,169.936300,-754.553300,-91.472712,-88.665219,-178.527919
C00643=1769.643700,173.179300,-754.553300,-91.472712,-88.665219,-178.527919
C00644=1769.715800,178.533800,-754.553300,-91.472712,-88.665219,-178.527919
C00645=1769.631500,179.950400,-754.553300,-91.472712,-88.665219,-178.527919
C00646=1769.720300,184.972100,-754.553300,-91.472712,-88.665219,-178.527919
C00647=1769.796000,188.294200,-754.553300,-91.472712,-88.665219,-178.527919
C00648=1769.878900,191.030400,-754.553300,-91.472712,-88.665219,-178.527919
C00649=1770.099900,194.160200,-754.553300,-91.472712,-88.665219,-178.527919
C00650=1770.015600,198.035900,-754.553300,-91.472712,-88.665219,-178.527919
C00651=1769.894600,201.520500,-754.553300,-91.472712,-88.665219,-178.527919
C00652=1770.071700,205.130700,-754.553300,-91.472712,-88.665219,-178.527919
C00653=1770.204500,210.053800,-754.553300,-91.472712,-88.665219,-178.527919
C00654=1770.042700,212.649100,-754.553300,-91.472712,-88.665219,-178.527919
C00655=1770.226400,217.953000,-754.553300,-91.472712,-88.665219,-178.527919
C00656=1770.237900,219.256100,-754.553300,-91.472712,-88.665219,-178.527919
C00657=1770.189100,223.508200,-754.553300,-91.472712,-88.665219,-178.527919
C00658=1770.301500,225.080200,-754.553300,-91.472712,-88.665219,-178.527919
C00659=1770.480400,228.239300,-754.553300,-91.472712,-88.665219,-178.527919
C00660=1770.466200,229.587400,-754.553300,-91.472712,-88.665219,-178.527919
C00661=1770.467400,232.993200,-754.553300,-91.472712,-88.665219,-178.527919
C00662=1770.521600,236.209500,-754.553300,-91.472712,-88.665219,-178.527919
C00663=1770.871600,237.577800,-754.553300,-91.472712,-88.665219,-178.527919
C00664=1770.844400,237.462900,-804.553300,-91.472712,-88.665219,-178.527919
C00665=1770.723800,236.493000,-804.553300,-91.472712,-88.665219,-178.527919
C00666=1770.337300,233.778700,-804.553300,-91.472712,-88.665219,-178.527919
C00667=1770.355400,231.488800,-804.553300,-91.472712,-88.665219,-178.527919
C00668=1770.369900,227.773100,-804.553300,-91.472712,-88.665219,-178.527919
C00669=1770.358200,225.823800,-804.553300,-91.472712,-88.665219,-178.527919
C00670=1770.350400,224.499000,-804.553300,-91.472712,-88.665219,-178.527919
C00671=1770.210700,220.390200,-804.553300,-91.472712,-88.665219,-178.527919
C00672=1770.207600,217.071500,-804.553300,-91.472712,-88.665219,-178.527919
C00673=1770.347400,212.570100,-804.553300,-91.472712,-88.665219,-178.527919
C00674=1770.222900,209.765300,-804.553300,-91.472712,-88.665219,-178.527919
C00675=1770.290600,206.580700,-804.553300,-91.472712,-88.665219,-178.527919
C00676=1770.239000,203.104600,-804.553300,-91.472712,-88.665219,-178.527919
C00677=1770.384300,201.611700,-804.553300,-91.472712,-88.665219,-178.527919
C00678=1770.259500,197.390700,-804.553300,-91.472712,-88.665219,-178.527919
C00679=1769.960000,193.357600,-804.553300,-91.472712,-88.665219,-178.527919
C00680=1770.210000,191.613800,-804.553300,-91.472712,-88.665219,-178.527919
C00681=1769.935000,187.131000,-804.553300,-91.472712,-88.665219,-178.527919
C00682=1769.947900,185.689700,-804.553300,-91.472712,-88.665219,-178.527919
C00683=1770.181100,182.756200,-804.553300,-91.472712,-88.665219,-178.527919
C00684=1769.882400,178.735500,-804.553300,-91.472712,-88.665219,-178.527919
C00685=1770.048700,173.534700,-804.553300,-91.472712,-88.665219,-178.527919
C00686=1770.113800,172.601900,-804.553300,-91.472712,-88.665219,-178.527919
C00687=1769.879300,168.707700,-804.553300,-91.472712,-88.665219,-178.527919
C00688=1770.082100,166.001700,-804.553300,-91.472712,-88.665219,-178.527919
C00689=1770.084900,162.513100,-804.553300,-91.472712,-88.665219,-178.527919
C00690=1769.963300,159.927900,-804.553300,-91.472712,-88.665219,-178.527919
C00691=1769.663900,157.209600,-804.553300,-91.472712,-88.665219,-178.527919
C00692=1770.144200,152.762900,-804.553300,-91.472712,-88.665219,-178.527919
C00693=1769.672600,148.605500,-804.553300,-91.472712,-88.665219,-178.527919
C00694=1769.839200,146.124900,-804.553300,-91.472712,-88.665219,-178.527919
C00695=1769.725200,142.027500,-804.553300,-91.472712,-88.665219,-178.527919
C00696=1769.824600,137.691600,-804.553300,-91.472712,-88.665219,-178.527919
C00697=1769.997800,134.235700,-804.553300,-91.472712,-88.665219,-178.527919
C00698=1769.937100,131.662000,-804.553300,-91.472712,-88.665219,-178.527919
C00699=1770.038200,127.889000,-804.553300,-91.472712,-88.665219,-178.527919
C00700=1770.213900,125.087200,-804.553300,-91.472712,-88.665219,-178.527919
C00701=1769.569100,120.835400,-804.553300,-91.472712,-88.665219,-178.527919
C00702=1769.587200,117.274900,-804.553300,-91.472712,-88.665219,-178.527919
C00703=1769.807000,113.172600,-804.553300,-91.472712,-88.665219,-178.527919
C00704=1769.913400,109.466600,-804.553300,-91.472712,-88.665219,-178.527919
C00705=1769.459600,107.326000,-804.553300,-91.472712,-88.665219,-178.527919
C00706=1769.572200,102.673200,-804.553300,-91.472712,-88.665219,-178.527919
C00707=1769.370100,98.743700,-804.553300,-91.472712,-88.665219,-178.527919
C00708=1769.572200,95.168200,-804.553300,-91.472712,-88.665219,-178.527919
C00709=1769.230300,91.353000,-804.553300,-91.472712,-88.665219,-178.527919
C00710=1769.804300,87.832300,-804.553300,-91.472712,-88.665219,-178.527919
C00711=1769.443800,83.087500,-804.553300,-91.472712,-88.665219,-178.527919
C00712=1769.497300,80.294600,-804.553300,-91.472712,-88.665219,-178.527919
C00713=1769.811700,76.747200,-804.553300,-91.472712,-88.665219,-178.527919
C00714=1769.038600,73.705900,-804.553300,-91.472712,-88.665219,-178.527919
C00715=1768.818000,70.211500,-804.553300,-91.472712,-88.665219,-178.527919
C00716=1769.160200,66.315300,-804.553300,-91.472712,-88.665219,-178.527919
C00717=1768.856300,64.063900,-804.553300,-91.472712,-88.665219,-178.527919
C00718=1769.613700,60.431500,-804.553300,-91.472712,-88.665219,-178.527919
C00719=1768.573600,58.458700,-804.553300,-91.472712,-88.665219,-178.527919
C00720=1768.649300,53.690100,-804.553300,-91.472712,-88.665219,-178.527919
C00721=1768.953900,50.364500,-804.553300,-91.472712,-88.665219,-178.527919
C00722=1769.005100,47.471100,-804.553300,-91.472712,-88.665219,-178.527919
C00723=1768.298300,43.158900,-804.553300,-91.472712,-88.665219,-178.527919
C00724=1768.828400,41.936300,-804.553300,-91.472712,-88.665219,-178.527919
C00725=1768.541700,38.874400,-804.553300,-91.472712,-88.665219,-178.527919
C00726=1769.349100,32.905900,-804.553300,-91.472712,-88.665219,-178.527919
C00727=1768.884900,30.966700,-804.553300,-91.472712,-88.665219,-178.527919
C00728=1769.245800,27.450500,-804.553300,-91.472712,-88.665219,-178.527919
C00729=1769.267600,23.511900,-804.553300,-91.472712,-88.665219,-178.527919
C00730=1768.171800,19.316700,-804.553300,-91.472712,-88.665219,-178.527919
C00731=1768.269700,15.837700,-804.553300,-91.472712,-88.665219,-178.527919
C00732=1768.146300,12.458500,-804.553300,-91.472712,-88.665219,-178.527919
C00733=1768.723500,8.023200,-804.553300,-91.472712,-88.665219,-178.527919
C00734=1768.551000,4.210300,-804.553300,-91.472712,-88.665219,-178.527919
C00735=1768.762200,1.323700,-804.553300,-91.472712,-88.665219,-178.527919
C00736=1768.826300,-1.567500,-804.553300,-91.472712,-88.665219,-178.527919
C00737=1768.448000,-5.947400,-804.553300,-91.472712,-88.665219,-178.527919
C00738=1767.963300,-10.150500,-804.553300,-91.472712,-88.665219,-178.527919
C00739=1768.177700,-12.752800,-804.553300,-91.472712,-88.665219,-178.527919
C00740=1767.742300,-16.059500,-804.553300,-91.472712,-88.665219,-178.527919
C00741=1768.556200,-20.772400,-804.553300,-91.472712,-88.665219,-178.527919
C00742=1768.931200,-22.547100,-804.553300,-91.472712,-88.665219,-178.527919
C00743=1767.704000,-26.308000,-804.553300,-91.472712,-88.665219,-178.527919
C00744=1767.538100,-30.938900,-804.553300,-91.472712,-88.665219,-178.527919
C00745=1767.429700,-32.774700,-804.553300,-91.472712,-88.665219,-178.527919
C00746=1768.717900,-36.731600,-804.553300,-91.472712,-88.665219,-178.527919
C00747=1767.732900,-39.421500,-804.553300,-91.472712,-88.665219,-178.527919
C00748=1767.404600,-45.117300,-804.553300,-91.472712,-88.665219,-178.527919
C00749=1767.493100,-48.250800,-804.553300,-91.472712,-88.665219,-178.527919
C00750=1767.962300,-51.101900,-804.553300,-91.472712,-88.665219,-178.527919
C00751=1768.710600,-54.210700,-804.553300,-91.472712,-88.665219,-178.527919
C00752=1768.057800,-57.684800,-804.553300,-91.472712,-88.665219,-178.527919
C00753=1767.702600,-61.333500,-804.553300,-91.472712,-88.665219,-178.527919
C00754=1767.678600,-64.475800,-804.553300,-91.472712,-88.665219,-178.527919
C00755=1768.407700,-67.120800,-804.553300,-91.472712,-88.665219,-178.527919
C00756=1767.521400,-72.013900,-804.553300,-91.472712,-88.665219,-178.527919
C00757=1767.378100,-75.083500,-804.553300,-91.472712,-88.665219,-178.527919
C00758=1768.297600,-78.262000,-804.553300,-91.472712,-88.665219,-178.527919
C00759=1768.343900,-83.043200,-804.553300,-91.472712,-88.665219,-178.527919
C00760=1767.751400,-86.562500,-804.553300,-91.472712,-88.665219,-178.527919
C00761=1767.818300,-89.417000,-804.553300,-91.472712,-88.665219,-178.527919
C00762=1767.775100,-94.557600,-804.553300,-91.472712,-88.665219,-178.527919
C00763=1767.577800,-96.727300,-804.553300,-91.472712,-88.665219,-178.527919
C00764=1768.020500,-101.050000,-804.553300,-91.472712,-88.665219,-178.527919
C00765=1768.317800,-103.238900,-804.553300,-91.472712,-88.665219,-178.527919
C00766=1768.355400,-107.465400,-804.553300,-91.472712,-88.665219,-178.527919
C00767=1767.931600,-111.484100,-804.553300,-91.472712,-88.665219,-178.527919
C00768=1768.365900,-114.876400,-804.553300,-91.472712,-88.665219,-178.527919
C00769=1767.992300,-118.251100,-804.553300,-91.472712,-88.665219,-178.527919
C00770=1768.559300,-122.022500,-804.553300,-91.472712,-88.665219,-178.527919
C00771=1768.274200,-125.666200,-804.553300,-91.472712,-88.665219,-178.527919
C00772=1768.281500,-129.300400,-804.553300,-91.472712,-88.665219,-178.527919
C00773=1768.701500,-132.752500,-804.553300,-91.472712,-88.665219,-178.527919
C00774=1768.379700,-136.376600,-804.553300,-91.472712,-88.665219,-178.527919
C00775=1768.668800,-141.236500,-804.553300,-91.472712,-88.665219,-178.527919
C00776=1768.904400,-144.706500,-804.553300,-91.472712,-88.665219,-178.527919
C00777=1768.725600,-148.991100,-804.553300,-91.472712,-88.665219,-178.527919
C00778=1768.873000,-150.838700,-804.553300,-91.472712,-88.665219,-178.527919
C00779=1768.856600,-154.828000,-804.553300,-91.472712,-88.665219,-178.527919
C00780=1768.617200,-157.537500,-804.553300,-91.472712,-88.665219,-178.527919
C00781=1768.733600,-159.966000,-804.553300,-91.472712,-88.665219,-178.527919
C00782=1769.659000,-160.358600,-854.553300,-91.472712,-88.665219,-178.527919
C00783=1769.379000,-159.416400,-854.553300,-91.472712,-88.665219,-178.527919
C00784=1769.258200,-157.507500,-854.553300,-91.472712,-88.665219,-178.527919
C00785=1769.399000,-153.993500,-854.553300,-91.472712,-88.665219,-178.527919
C00786=1769.464500,-150.232600,-854.553300,-91.472712,-88.665219,-178.527919
C00787=1769.018000,-147.624900,-854.553300,-91.472712,-88.665219,-178.527919
C00788=1769.248200,-145.633700,-854.553300,-91.472712,-88.665219,-178.527919
C00789=1769.288500,-140.819900,-854.553300,-91.472712,-88.665219,-178.527919
C00790=1768.999500,-136.296800,-854.553300,-91.472712,-88.665219,-178.527919
C00791=1768.827700,-132.387100,-854.553300,-91.472712,-88.665219,-178.527919
C00792=1769.504600,-126.692500,-854.553300,-91.472712,-88.665219,-178.527919
C00793=1769.743300,-122.232000,-854.553300,-91.472712,-88.665219,-178.527919
C00794=1769.748900,-118.661900,-854.553300,-91.472712,-88.665219,-178.527919
C00795=1768.638100,-116.438900,-854.553300,-91.472712,-88.665219,-178.527919
C00796=1769.434900,-112.700300,-854.553300,-91.472712,-88.665219,-178.527919
C00797=1768.612300,-110.474200,-854.553300,-91.472712,-88.665219,-178.527919
C00798=1769.880000,-107.423200,-854.553300,-91.472712,-88.665219,-178.527919
C00799=1768.754200,-104.411600,-854.553300,-91.472712,-88.665219,-178.527919
C00800=1769.087000,-100.363500,-854.553300,-91.472712,-88.665219,-178.527919
C00801=1768.834300,-96.404000,-854.553300,-91.472712,-88.665219,-178.527919
C00802=1769.501100,-92.644400,-854.553300,-91.472712,-88.665219,-178.527919
C00803=1769.120100,-90.945700,-854.553300,-91.472712,-88.665219,-178.527919
C00804=1769.924200,-87.567900,-854.553300,-91.472712,-88.665219,-178.527919
C00805=1769.414300,-82.448900,-854.553300,-91.472712,-88.665219,-178.527919
C00806=1769.561400,-78.856600,-854.553300,-91.472712,-88.665219,-178.527919
C00807=1769.709900,-74.058200,-854.553300,-91.472712,-88.665219,-178.527919
C00808=1769.743700,-73.149400,-854.553300,-91.472712,-88.665219,-178.527919
C00809=1768.877200,-70.289800,-854.553300,-91.472712,-88.665219,-178.527919
C00810=1768.295100,-65.471800,-854.553300,-91.472712,-88.665219,-178.527919
C00811=1768.654100,-61.404500,-854.553300,-91.472712,-88.665219,-178.527919
C00812=1769.007900,-56.895600,-854.553300,-91.472712,-88.665219,-178.527919
C00813=1769.567300,-54.540100,-854.553300,-91.472712,-88.665219,-178.527919
C00814=1769.720000,-49.794700,-854.553300,-91.472712,-88.665219,-178.527919
C00815=1768.743000,-46.454800,-854.553300,-91.472712,-88.665219,-178.527919
C00816=1770.441800,-43.231100,-854.553300,-91.472712,-88.665219,-178.527919
C00817=1770.058100,-42.064500,-854.553300,-91.472712,-88.665219,-178.527919
C00818=1770.391300,-37.632600,-854.553300,-91.472712,-88.665219,-178.527919
C00819=1770.110400,-36.165200,-854.553300,-91.472712,-88.665219,-178.527919
C00820=1769.610900,-32.947400,-854.553300,-91.472712,-88.665219,-178.527919
C00821=1768.851400,-30.837900,-854.553300,-91.472712,-88.665219,-178.527919
C00822=1769.201400,-26.343100,-854.553300,-91.472712,-88.665219,-178.527919
C00823=1770.435900,-23.262700,-854.553300,-91.472712,-88.665219,-178.527919
C00824=1769.770500,-18.058100,-854.553300,-91.472712,-88.665219,-178.527919
C00825=1769.552000,-15.022600,-854.553300,-91.472712,-88.665219,-178.527919
C00826=1770.571800,-8.367000,-854.553300,-91.472712,-88.665219,-178.527919
C00827=1769.058500,-7.188300,-854.553300,-91.472712,-88.665219,-178.527919
C00828=1769.395800,-2.772000,-854.553300,-91.472712,-88.665219,-178.527919
C00829=1769.385000,1.187200,-854.553300,-91.472712,-88.665219,-178.527919
C00830=1770.594100,6.646600,-854.553300,-91.472712,-88.665219,-178.527919
C00831=1769.832900,10.862200,-854.553300,-91.472712,-88.665219,-178.527919
C00832=1769.816200,14.588700,-854.553300,-91.472712,-88.665219,-178.527919
C00833=1770.803300,17.863000,-854.553300,-91.472712,-88.665219,-178.527919
C00834=1769.969600,22.078900,-854.553300,-91.472712,-88.665219,-178.527919
C00835=1770.646400,26.469800,-854.553300,-91.472712,-88.665219,-178.527919
C00836=1769.712300,30.118600,-854.553300,-91.472712,-88.665219,-178.527919
C00837=1770.019400,33.396800,-854.553300,-91.472712,-88.665219,-178.527919
C00838=1770.546000,38.068500,-854.553300,-91.472712,-88.665219,-178.527919
C00839=1770.852400,41.878000,-854.553300,-91.472712,-88.665219,-178.527919
C00840=1769.841300,45.608000,-854.553300,-91.472712,-88.665219,-178.527919
C00841=1770.582600,47.255800,-854.553300,-91.472712,-88.665219,-178.527919
C00842=1770.469400,52.058600,-854.553300,-91.472712,-88.665219,-178.527919
C00843=1769.885900,53.858100,-854.553300,-91.472712,-88.665219,-178.527919
C00844=1770.812000,57.250300,-854.553300,-91.472712,-88.665219,-178.527919
C00845=1770.296100,61.976700,-854.553300,-91.472712,-88.665219,-178.527919
C00846=1770.568000,67.372200,-854.553300,-91.472712,-88.665219,-178.527919
C00847=1769.936800,70.633500,-854.553300,-91.472712,-88.665219,-178.527919
C00848=1770.239000,74.008600,-854.553300,-91.472712,-88.665219,-178.527919
C00849=1770.924900,77.011000,-854.553300,-91.472712,-88.665219,-178.527919
C00850=1770.594500,81.420300,-854.553300,-91.472712,-88.665219,-178.527919
C00851=1770.813700,85.166700,-854.553300,-91.472712,-88.665219,-178.527919
C00852=1770.982400,88.354600,-854.553300,-91.472712,-88.665219,-178.527919
C00853=1770.248400,92.142200,-854.553300,-91.472712,-88.665219,-178.527919
C00854=1770.068700,94.517900,-854.553300,-91.472712,-88.665219,-178.527919
C00855=1770.543600,98.786600,-854.553300,-91.472712,-88.665219,-178.527919
C00856=1770.846100,101.859600,-854.553300,-91.472712,-88.665219,-178.527919
C00857=1770.385700,105.490800,-854.553300,-91.472712,-88.665219,-178.527919
C00858=1769.979000,108.244200,-854.553300,-91.472712,-88.665219,-178.527919
C00859=1770.703600,111.835500,-854.553300,-91.472712,-88.665219,-178.527919
C00860=1770.358900,115.867400,-854.553300,-91.472712,-88.665219,-178.527919
C00861=1770.278000,118.383700,-854.553300,-91.472712,-88.665219,-178.527919
C00862=1770.449200,122.523300,-854.553300,-91.472712,-88.665219,-178.527919
C00863=1770.503500,127.262900,-854.553300,-91.472712,-88.665219,-178.527919
C00864=1770.488900,129.265700,-854.553300,-91.472712,-88.665219,-178.527919
C00865=1770.922800,133.347400,-854.553300,-91.472712,-88.665219,-178.527919
C00866=1770.385000,137.018900,-854.553300,-91.472712,-88.665219,-178.527919
C00867=1770.438300,138.481800,-854.553300,-91.472712,-88.665219,-178.527919
C00868=1770.381200,142.576200,-854.553300,-91.472712,-88.665219,-178.527919
C00869=1770.454700,147.052300,-854.553300,-91.472712,-88.665219,-178.527919
C00870=1770.132300,150.544900,-854.553300,-91.472712,-88.665219,-178.527919
C00871=1770.423000,153.424400,-854.553300,-91.472712,-88.665219,-178.527919
C00872=1770.556900,159.242100,-854.553300,-91.472712,-88.665219,-178.527919
C00873=1770.523700,163.941200,-854.553300,-91.472712,-88.665219,-178.527919
C00874=1770.466200,167.171000,-854.553300,-91.472712,-88.665219,-178.527919
C00875=1770.306200,173.946200,-854.553300,-91.472712,-88.665219,-178.527919
C00876=1770.826600,177.980700,-854.553300,-91.472712,-88.665219,-178.527919
C00877=1770.508400,180.304800,-854.553300,-91.472712,-88.665219,-178.527919
C00878=1770.527900,184.291000,-854.553300,-91.472712,-88.665219,-178.527919
C00879=1770.799800,187.711700,-854.553300,-91.472712,-88.665219,-178.527919
C00880=1770.749200,191.665500,-854.553300,-91.472712,-88.665219,-178.527919
C00881=1770.393700,194.037200,-854.553300,-91.472712,-88.665219,-178.527919
C00882=1770.451200,198.269100,-854.553300,-91.472712,-88.665219,-178.527919
C00883=1770.421300,200.573200,-854.553300,-91.472712,-88.665219,-178.527919
C00884=1770.318800,203.787800,-854.553300,-91.472712,-88.665219,-178.527919
C00885=1770.324400,208.027100,-854.553300,-91.472712,-88.665219,-178.527919
C00886=1770.528300,211.453800,-854.553300,-91.472712,-88.665219,-178.527919
C00887=1770.333400,215.077200,-854.553300,-91.472712,-88.665219,-178.527919
C00888=1770.355200,218.525000,-854.553300,-91.472712,-88.665219,-178.527919
C00889=1770.813000,223.342500,-854.553300,-91.472712,-88.665219,-178.527919
C00890=1770.446000,224.446400,-854.553300,-91.472712,-88.665219,-178.527919
C00891=1770.642700,227.782000,-854.553300,-91.472712,-88.665219,-178.527919
C00892=1770.488400,229.172500,-854.553300,-91.472712,-88.665219,-178.527919
C00893=1770.289500,233.314200,-854.553300,-91.472712,-88.665219,-178.527919
C00894=1770.516800,235.381400,-854.553300,-91.472712,-88.665219,-178.527919
C00895=1770.587900,237.600400,-854.553300,-91.472712,-88.665219,-178.527919
C00896=1795.634000,216.962000,-456.179300,-176.322032,-0.120321,-90.000210
C00897=1801.219000,216.962000,-456.521300,-176.322032,-0.120321,-90.000210
C00898=1802.338900,216.962000,-456.827000,-176.322032,-0.120321,-90.000210
C00899=1806.351700,216.962000,-456.685400,-176.322032,-0.120321,-90.000210
C00900=1807.197200,216.962000,-456.858700,-176.322032,-0.120321,-90.000210
C00901=1811.407300,216.962000,-457.126500,-176.322032,-0.120321,-90.000210
C00902=1812.062900,216.962000,-457.033100,-176.322032,-0.120321,-90.000210
C00903=1817.500600,216.962000,-457.407600,-176.322032,-0.120321,-90.000210
C00904=1818.193000,216.962000,-456.864900,-176.322032,-0.120321,-90.000210
C00905=1821.847300,216.962000,-457.041800,-176.322032,-0.120321,-90.000210
C00906=1824.852500,216.962000,-457.294300,-176.322032,-0.120321,-90.000210
C00907=1826.988500,216.962000,-457.252300,-176.322032,-0.120321,-90.000210
C00908=1830.848800,216.962000,-457.515600,-176.322032,-0.120321,-90.000210
C00909=1831.812600,216.962000,-457.618300,-176.322032,-0.120321,-90.000210
C00910=1836.392800,216.962000,-457.452900,-176.322032,-0.120321,-90.000210
C00911=1837.826000,216.962000,-457.911000,-176.322032,-0.120321,-90.000210
C00912=1841.442300,216.962000,-457.245900,-176.322032,-0.120321,-90.000210
C00913=1843.603300,216.962000,-458.036300,-176.322032,-0.120321,-90.000210
C00914=1846.357400,216.962000,-458.131600,-176.322032,-0.120321,-90.000210
C00915=1851.492800,216.962000,-457.681100,-176.322032,-0.120321,-90.000210
C00916=1852.150000,216.962000,-458.603400,-176.322032,-0.120321,-90.000210
C00917=1856.218500,216.962000,-457.936700,-176.322032,-0.120321,-90.000210
C00918=1857.510900,216.962000,-457.609800,-176.322032,-0.120321,-90.000210
C00919=1861.892200,216.962000,-457.735500,-176.322032,-0.120321,-90.000210
C00920=1863.181000,216.962000,-457.900100,-176.322032,-0.120321,-90.000210
C00921=1867.366500,216.962000,-458.477300,-176.322032,-0.120321,-90.000210
C00922=1871.813400,216.962000,-457.443600,-176.322032,-0.120321,-90.000210
C00923=1872.445500,216.962000,-457.772700,-176.322032,-0.120321,-90.000210
C00924=1876.439100,216.962000,-459.417200,-176.322032,-0.120321,-90.000210
C00925=1877.286900,216.962000,-458.047200,-176.322032,-0.120321,-90.000210
C00926=1881.612800,216.962000,-458.097500,-176.322032,-0.120321,-90.000210
C00927=1882.550000,216.962000,-459.273400,-176.322032,-0.120321,-90.000210
C00928=1886.540700,216.962000,-459.690500,-176.322032,-0.120321,-90.000210
C00929=1890.633900,216.962000,-458.464900,-176.322032,-0.120321,-90.000210
C00930=1891.646700,216.962000,-458.348800,-176.322032,-0.120321,-90.000210
C00931=1895.894700,216.962000,-459.385500,-176.322032,-0.120321,-90.000210
C00932=1896.783800,216.962000,-458.593800,-176.322032,-0.120321,-90.000210
C00933=1901.744400,216.962000,-459.089300,-176.322032,-0.120321,-90.000210
C00934=1902.841100,216.962000,-459.487400,-176.322032,-0.120321,-90.000210
C00935=1906.630900,216.962000,-458.457100,-176.322032,-0.120321,-90.000210
C00936=1908.829300,216.962000,-460.090400,-176.322032,-0.120321,-90.000210
C00937=1911.722800,216.962000,-459.615500,-176.322032,-0.120321,-90.000210
C00938=1917.025800,216.962000,-458.838500,-176.322032,-0.120321,-90.000210
C00939=1917.470100,216.962000,-460.228700,-176.322032,-0.120321,-90.000210
C00940=1921.109200,216.962000,-457.818700,-176.322032,-0.120321,-90.000210
C00941=1923.007900,216.962000,-459.438200,-176.322032,-0.120321,-90.000210
C00942=1926.358200,216.962000,-457.783100,-176.322032,-0.120321,-90.000210
C00943=1927.995900,216.962000,-459.776800,-176.322032,-0.120321,-90.000210
C00944=1931.743700,216.962000,-458.553100,-176.322032,-0.120321,-90.000210
C00945=1934.407300,216.962000,-459.389100,-176.322032,-0.120321,-90.000210
C00946=1936.432400,216.962000,-457.544300,-176.322032,-0.120321,-90.000210
C00947=1940.623800,216.962000,-458.235300,-176.322032,-0.120321,-90.000210
C00948=1941.931000,216.962000,-460.394700,-176.322032,-0.120321,-90.000210
C00949=1946.079500,216.962000,-459.120400,-176.322032,-0.120321,-90.000210
C00950=1947.288700,216.962000,-458.765300,-176.322032,-0.120321,-90.000210
C00951=1951.448200,216.962000,-459.871800,-176.322032,-0.120321,-90.000210
C00952=1952.709600,216.962000,-458.082100,-176.322032,-0.120321,-90.000210
C00953=1956.590000,216.962000,-458.255200,-176.322032,-0.120321,-90.000210
C00954=1958.150200,216.962000,-458.551500,-176.322032,-0.120321,-90.000210
C00955=1962.188200,216.962000,-458.115300,-176.322032,-0.120321,-90.000210
C00956=1965.761500,216.962000,-460.136000,-176.322032,-0.120321,-90.000210
C00957=1966.901900,216.962000,-457.751500,-176.322032,-0.120321,-90.000210
C00958=1970.875400,216.962000,-459.753000,-176.322032,-0.120321,-90.000210
C00959=1972.098300,216.962000,-459.851200,-176.322032,-0.120321,-90.000210
C00960=1975.958500,216.962000,-459.061000,-176.322032,-0.120321,-90.000210
C00961=1977.447800,216.962000,-459.489400,-176.322032,-0.120321,-90.000210
C00962=1981.499100,216.962000,-459.739600,-176.322032,-0.120321,-90.000210
C00963=1982.799900,216.962000,-458.905300,-176.322032,-0.120321,-90.000210
C00964=1986.506900,216.962000,-458.530200,-176.322032,-0.120321,-90.000210
C00965=1987.289200,216.962000,-456.746100,-176.322032,-0.120321,-90.000210
C00966=1991.003400,216.962000,-459.603800,-176.322032,-0.120321,-90.000210
C00967=1992.224700,216.962000,-456.666300,-176.322032,-0.120321,-90.000210
C00968=1996.817800,216.962000,-458.372300,-176.322032,-0.120321,-90.000210
C00969=1997.523200,216.962000,-459.384500,-176.322032,-0.120321,-90.000210
C00970=2002.179300,216.962000,-458.668200,-176.322032,-0.120321,-90.000210
C00971=2004.158100,216.962000,-458.937300,-176.322032,-0.120321,-90.000210
C00972=2007.098900,216.962000,-458.477700,-176.322032,-0.120321,-90.000210
C00973=2010.420400,216.962000,-457.773000,-176.322032,-0.120321,-90.000210
C00974=2012.306300,216.962000,-458.927400,-176.322032,-0.120321,-90.000210
C00975=2016.056400,216.962000,-459.400600,-176.322032,-0.120321,-90.000210
C00976=2016.909300,216.962000,-458.358100,-176.322032,-0.120321,-90.000210
C00977=2020.788700,216.962000,-458.796100,-176.322032,-0.120321,-90.000210
C00978=2021.854200,216.962000,-458.003900,-176.322032,-0.120321,-90.000210
C00979=2025.872500,216.962000,-458.489000,-176.322032,-0.120321,-90.000210
C00980=2026.895500,216.962000,-456.503700,-176.322032,-0.120321,-90.000210
C00981=2031.392000,216.962000,-458.334900,-176.322032,-0.120321,-90.000210
C00982=2032.597200,216.962000,-458.628900,-176.322032,-0.120321,-90.000210
C00983=2037.476800,216.962000,-458.297700,-176.322032,-0.120321,-90.000210
C00984=2038.952300,216.962000,-458.864600,-176.322032,-0.120321,-90.000210
C00985=2042.233300,216.962000,-458.621200,-176.322032,-0.120321,-90.000210
C00986=2042.967700,216.962000,-459.442400,-176.322032,-0.120321,-90.000210
C00987=2046.399400,216.962000,-458.298000,-176.322032,-0.120321,-90.000210
C00988=2051.148500,216.962000,-457.982900,-176.322032,-0.120321,-90.000210
C00989=2052.154900,216.962000,-458.313700,-176.322032,-0.120321,-90.000210
C00990=2056.928600,216.962000,-456.750300,-176.322032,-0.120321,-90.000210
C00991=2057.982400,216.962000,-459.654200,-176.322032,-0.120321,-90.000210
C00992=2061.792000,216.962000,-457.960400,-176.322032,-0.120321,-90.000210
C00993=2062.613500,216.962000,-458.560000,-176.322032,-0.120321,-90.000210
C00994=2066.755800,216.962000,-457.209500,-176.322032,-0.120321,-90.000210
C00995=2069.307600,216.962000,-458.258700,-176.322032,-0.120321,-90.000210
C00996=2072.075600,216.962000,-458.227000,-176.322032,-0.120321,-90.000210
C00997=2076.450300,216.962000,-457.622800,-176.322032,-0.120321,-90.000210
C00998=2077.214400,216.962000,-458.644800,-176.322032,-0.120321,-90.000210
C00999=2081.235200,216.962000,-458.164300,-176.322032,-0.120321,-90.000210
C01000=2081.828100,216.962000,-456.135200,-176.322032,-0.120321,-90.000210
C01001=2086.144000,216.962000,-457.836300,-176.322032,-0.120321,-90.000210
C01002=2087.140300,216.962000,-456.091300,-176.322032,-0.120321,-90.000210
C01003=2090.435100,216.962000,-457.540400,-176.322032,-0.120321,-90.000210
C01004=2092.517400,216.962000,-457.453500,-176.322032,-0.120321,-90.000210
C01005=2096.814200,216.962000,-457.433500,-176.322032,-0.120321,-90.000210
C01006=2097.456700,216.962000,-456.346600,-176.322032,-0.120321,-90.000210
C01007=2101.142400,216.962000,-456.017300,-176.322032,-0.120321,-90.000210
C01008=2102.030300,216.962000,-458.063200,-176.322032,-0.120321,-90.000210
C01009=2106.556100,216.962000,-456.905100,-176.322032,-0.120321,-90.000210
C01010=2107.182200,216.962000,-457.894500,-176.322032,-0.120321,-90.000210
C01011=2111.481200,216.962000,-457.141800,-176.322032,-0.120321,-90.000210
C01012=2112.120900,216.962000,-456.228700,-176.322032,-0.120321,-90.000210
C01013=2115.864300,216.962000,-456.737100,-176.322032,-0.120321,-90.000210
C01014=2117.634900,216.962000,-456.543200,-176.322032,-0.120321,-90.000210
C01015=2118.826200,216.962000,-456.984400,-176.322032,-0.120321,-90.000210
C01016=2121.655300,216.962000,-456.933700,-176.322032,-0.120321,-90.000210
C01017=2123.613800,216.962000,-455.976200,-176.322032,-0.120321,-90.000210
C01018=2126.454900,216.962000,-457.351400,-176.322032,-0.120321,-90.000210
C01019=2127.300700,216.962000,-457.090500,-176.322032,-0.120321,-90.000210
C01020=2132.055200,216.962000,-456.168200,-176.322032,-0.120321,-90.000210
C01021=2134.405800,216.962000,-455.803300,-176.322032,-0.120321,-90.000210
C01022=2137.204100,216.962000,-456.231100,-176.322032,-0.120321,-90.000210
C01023=2138.787100,216.962000,-455.771400,-176.322032,-0.120321,-90.000210
C01024=2141.568100,216.962000,-456.331800,-176.322032,-0.120321,-90.000210
C01025=2142.773700,216.962000,-456.551100,-176.322032,-0.120321,-90.000210
C01026=2146.144200,216.962000,-456.205800,-176.322032,-0.120321,-90.000210
C01027=2147.932900,216.962000,-456.281100,-176.322032,-0.120321,-90.000210
C01028=2151.187100,216.962000,-456.059000,-176.322032,-0.120321,-90.000210
C01029=2152.073000,216.962000,-456.166100,-176.322032,-0.120321,-90.000210
C01030=2153.314400,216.962000,-455.905400,-176.322032,-0.120321,-90.000210
C01031=2156.669700,216.962000,-456.070300,-176.322032,-0.120321,-90.000210
C01032=2157.790100,216.962000,-456.167600,-176.322032,-0.120321,-90.000210
C01033=2160.396500,216.962000,-456.482300,-176.322032,-0.120321,-90.000210
C01034=2161.718200,216.962000,-455.880700,-176.322032,-0.120321,-90.000210
C01035=2162.603500,216.962000,-455.884000,-176.322032,-0.120321,-90.000210
C01036=2165.564100,216.962000,-455.751600,-176.322032,-0.120321,-90.000210
C01037=2167.393800,216.962000,-455.756400,-176.322032,-0.120321,-90.000210
C01038=2167.831000,216.962000,-456.075000,-176.322032,-0.120321,-90.000210
C01039=2171.335100,216.962000,-456.118300,-176.322032,-0.120321,-90.000210
C01040=2172.435800,216.962000,-455.732000,-176.322032,-0.120321,-90.000210
C01041=2173.858700,216.962000,-456.094100,-176.322032,-0.120321,-90.000210
C01042=2176.131300,216.962000,-455.881700,-176.322032,-0.120321,-90.000210
C01043=2177.352600,216.962000,-456.067400,-176.322032,-0.120321,-90.000210
C01044=2179.816400,216.962000,-455.745000,-176.322032,-0.120321,-90.000210
C01045=2182.077000,216.962000,-455.258000,-176.322032,-0.120321,-90.000210
C01046=2185.611400,216.962000,-456.005800,-176.322032,-0.120321,-90.000210
C01047=2187.042800,216.962000,-455.530700,-176.322032,-0.120321,-90.000210
C01048=2188.010000,166.962000,-454.226400,-176.322032,-0.120321,-90.000210
C01049=2186.540100,166.962000,-454.377100,-176.322032,-0.120321,-90.000210
C01050=2182.393000,166.962000,-455.132100,-176.322032,-0.120321,-90.000210
C01051=2181.661100,166.962000,-455.821900,-176.322032,-0.120321,-90.000210
C01052=2177.839600,166.962000,-455.614800,-176.322032,-0.120321,-90.000210
C01053=2176.397900,166.962000,-456.103300,-176.322032,-0.120321,-90.000210
C01054=2175.381500,166.962000,-456.054900,-176.322032,-0.120321,-90.000210
C01055=2172.619000,166.962000,-455.720000,-176.322032,-0.120321,-90.000210
C01056=2172.194100,166.962000,-455.501700,-176.322032,-0.120321,-90.000210
C01057=2171.264400,166.962000,-456.175300,-176.322032,-0.120321,-90.000210
C01058=2169.184100,166.962000,-455.866200,-176.322032,-0.120321,-90.000210
C01059=2167.106700,166.962000,-455.923200,-176.322032,-0.120321,-90.000210
C01060=2166.513200,166.962000,-456.229100,-176.322032,-0.120321,-90.000210
C01061=2162.847400,166.962000,-456.452300,-176.322032,-0.120321,-90.000210
C01062=2162.074500,166.962000,-456.532200,-176.322032,-0.120321,-90.000210
C01063=2157.352100,166.962000,-456.507600,-176.322032,-0.120321,-90.000210
C01064=2156.469500,166.962000,-457.039800,-176.322032,-0.120321,-90.000210
C01065=2151.713600,166.962000,-456.601100,-176.322032,-0.120321,-90.000210
C01066=2150.868900,166.962000,-456.635400,-176.322032,-0.120321,-90.000210
C01067=2147.097400,166.962000,-457.175100,-176.322032,-0.120321,-90.000210
C01068=2145.643800,166.962000,-456.476700,-176.322032,-0.120321,-90.000210
C01069=2142.330000,166.962000,-457.905700,-176.322032,-0.120321,-90.000210
C01070=2141.518600,166.962000,-456.846800,-176.322032,-0.120321,-90.000210
C01071=2137.112600,166.962000,-458.006600,-176.322032,-0.120321,-90.000210
C01072=2136.030600,166.962000,-457.323200,-176.322032,-0.120321,-90.000210
C01073=2132.224300,166.962000,-458.198800,-176.322032,-0.120321,-90.000210
C01074=2131.462800,166.962000,-457.850200,-176.322032,-0.120321,-90.000210
C01075=2126.829500,166.962000,-457.183500,-176.322032,-0.120321,-90.000210
C01076=2126.294800,166.962000,-458.530600,-176.322032,-0.120321,-90.000210
C01077=2121.506000,166.962000,-457.738000,-176.322032,-0.120321,-90.000210
C01078=2120.636800,166.962000,-458.068600,-176.322032,-0.120321,-90.000210
C01079=2116.907500,166.962000,-458.671600,-176.322032,-0.120321,-90.000210
C01080=2116.115600,166.962000,-458.061000,-176.322032,-0.120321,-90.000210
C01081=2111.765500,166.962000,-458.760400,-176.322032,-0.120321,-90.000210
C01082=2110.603000,166.962000,-458.350200,-176.322032,-0.120321,-90.000210
C01083=2106.984500,166.962000,-458.780500,-176.322032,-0.120321,-90.000210
C01084=2105.997100,166.962000,-459.326200,-176.322032,-0.120321,-90.000210
C01085=2101.865600,166.962000,-458.047600,-176.322032,-0.120321,-90.000210
C01086=2101.266500,166.962000,-458.440500,-176.322032,-0.120321,-90.000210
C01087=2096.103400,166.962000,-458.806700,-176.322032,-0.120321,-90.000210
C01088=2095.255000,166.962000,-459.548700,-176.322032,-0.120321,-90.000210
C01089=2091.428200,166.962000,-459.755700,-176.322032,-0.120321,-90.000210
C01090=2089.390100,166.962000,-459.034800,-176.322032,-0.120321,-90.000210
C01091=2087.410400,166.962000,-459.721700,-176.322032,-0.120321,-90.000210
C01092=2085.989400,166.962000,-459.831000,-176.322032,-0.120321,-90.000210
C01093=2081.994000,166.962000,-458.736500,-176.322032,-0.120321,-90.000210
C01094=2081.443500,166.962000,-460.389100,-176.322032,-0.120321,-90.000210
C01095=2076.668000,166.962000,-459.982600,-176.322032,-0.120321,-90.000210
C01096=2075.991500,166.962000,-460.187500,-176.322032,-0.120321,-90.000210
C01097=2072.240100,166.962000,-458.962500,-176.322032,-0.120321,-90.000210
C01098=2070.271200,166.962000,-460.359500,-176.322032,-0.120321,-90.000210
C01099=2067.226000,166.962000,-459.812200,-176.322032,-0.120321,-90.000210
C01100=2066.468000,166.962000,-460.260700,-176.322032,-0.120321,-90.000210
C01101=2062.200200,166.962000,-460.024900,-176.322032,-0.120321,-90.000210
C01102=2061.092900,166.962000,-459.366900,-176.322032,-0.120321,-90.000210
C01103=2056.985200,166.962000,-460.955100,-176.322032,-0.120321,-90.000210
C01104=2055.799500,166.962000,-459.487200,-176.322032,-0.120321,-90.000210
C01105=2051.990700,166.962000,-459.979300,-176.322032,-0.120321,-90.000210
C01106=2051.341300,166.962000,-460.342800,-176.322032,-0.120321,-90.000210
C01107=2047.971800,166.962000,-460.187500,-176.322032,-0.120321,-90.000210
C01108=2046.536100,166.962000,-460.353200,-176.322032,-0.120321,-90.000210
C01109=2045.295600,166.962000,-460.944300,-176.322032,-0.120321,-90.000210
C01110=2042.137600,166.962000,-459.742300,-176.322032,-0.120321,-90.000210
C01111=2040.934300,166.962000,-460.912300,-176.322032,-0.120321,-90.000210
C01112=2036.887700,166.962000,-459.461000,-176.322032,-0.120321,-90.000210
C01113=2036.355600,166.962000,-460.110400,-176.322032,-0.120321,-90.000210
C01114=2035.001400,166.962000,-460.955800,-176.322032,-0.120321,-90.000210
C01115=2031.686000,166.962000,-460.027600,-176.322032,-0.120321,-90.000210
C01116=2031.299900,166.962000,-461.293600,-176.322032,-0.120321,-90.000210
C01117=2027.511500,166.962000,-461.044700,-176.322032,-0.120321,-90.000210
C01118=2026.516400,166.962000,-461.230100,-176.322032,-0.120321,-90.000210
C01119=2022.395300,166.962000,-459.873100,-176.322032,-0.120321,-90.000210
C01120=2021.679700,166.962000,-460.447800,-176.322032,-0.120321,-90.000210
C01121=2018.181500,166.962000,-460.348900,-176.322032,-0.120321,-90.000210
C01122=2016.721500,166.962000,-461.371200,-176.322032,-0.120321,-90.000210
C01123=2014.931300,166.962000,-460.141800,-176.322032,-0.120321,-90.000210
C01124=2012.761500,166.962000,-461.148100,-176.322032,-0.120321,-90.000210
C01125=2011.570600,166.962000,-459.842200,-176.322032,-0.120321,-90.000210
C01126=2007.788100,166.962000,-461.601700,-176.322032,-0.120321,-90.000210
C01127=2006.592300,166.962000,-459.982100,-176.322032,-0.120321,-90.000210
C01128=2005.922400,166.962000,-461.003400,-176.322032,-0.120321,-90.000210
C01129=2001.752300,166.962000,-460.634700,-176.322032,-0.120321,-90.000210
C01130=2000.631600,166.962000,-459.957800,-176.322032,-0.120321,-90.000210
C01131=1997.097500,166.962000,-460.993600,-176.322032,-0.120321,-90.000210
C01132=1996.283700,166.962000,-461.179200,-176.322032,-0.120321,-90.000210
C01133=1992.996700,166.962000,-460.238500,-176.322032,-0.120321,-90.000210
C01134=1992.223600,166.962000,-460.402800,-176.322032,-0.120321,-90.000210
C01135=1989.293700,166.962000,-460.890300,-176.322032,-0.120321,-90.000210
C01136=1986.959800,166.962000,-460.231000,-176.322032,-0.120321,-90.000210
C01137=1985.899600,166.962000,-461.410900,-176.322032,-0.120321,-90.000210
C01138=1981.731800,166.962000,-460.408400,-176.322032,-0.120321,-90.000210
C01139=1979.408700,166.962000,-461.264300,-176.322032,-0.120321,-90.000210
C01140=1976.846600,166.962000,-460.516600,-176.322032,-0.120321,-90.000210
C01141=1975.662700,166.962000,-460.790500,-176.322032,-0.120321,-90.000210
C01142=1973.210000,166.962000,-460.744100,-176.322032,-0.120321,-90.000210
C01143=1971.617300,166.962000,-461.263300,-176.322032,-0.120321,-90.000210
C01144=1970.920100,166.962000,-460.732200,-176.322032,-0.120321,-90.000210
C01145=1966.975600,166.962000,-461.559700,-176.322032,-0.120321,-90.000210
C01146=1966.068000,166.962000,-461.766000,-176.322032,-0.120321,-90.000210
C01147=1962.546900,166.962000,-460.398500,-176.322032,-0.120321,-90.000210
C01148=1961.215300,166.962000,-460.764500,-176.322032,-0.120321,-90.000210
C01149=1958.441900,166.962000,-460.653500,-176.322032,-0.120321,-90.000210
C01150=1956.874400,166.962000,-461.717600,-176.322032,-0.120321,-90.000210
C01151=1953.202900,166.962000,-460.752000,-176.322032,-0.120321,-90.000210
C01152=1951.501200,166.962000,-459.958400,-176.322032,-0.120321,-90.000210
C01153=1950.523000,166.962000,-461.648900,-176.322032,-0.120321,-90.000210
C01154=1946.804000,166.962000,-461.988500,-176.322032,-0.120321,-90.000210
C01155=1945.609500,166.962000,-461.853100,-176.322032,-0.120321,-90.000210
C01156=1942.208400,166.962000,-461.311200,-176.322032,-0.120321,-90.000210
C01157=1941.944000,166.962000,-462.089900,-176.322032,-0.120321,-90.000210
C01158=1938.817100,166.962000,-461.262700,-176.322032,-0.120321,-90.000210
C01159=1937.110100,166.962000,-461.285800,-176.322032,-0.120321,-90.000210
C01160=1933.825600,166.962000,-461.105300,-176.322032,-0.120321,-90.000210
C01161=1931.814800,166.962000,-462.065900,-176.322032,-0.120321,-90.000210
C01162=1930.239400,166.962000,-460.655800,-176.322032,-0.120321,-90.000210
C01163=1926.890500,166.962000,-462.327500,-176.322032,-0.120321,-90.000210
C01164=1926.103700,166.962000,-461.533800,-176.322032,-0.120321,-90.000210
C01165=1922.471700,166.962000,-461.141500,-176.322032,-0.120321,-90.000210
C01166=1921.270900,166.962000,-461.390100,-176.322032,-0.120321,-90.000210
C01167=1916.452300,166.962000,-461.084700,-176.322032,-0.120321,-90.000210
C01168=1916.288800,166.962000,-461.747800,-176.322032,-0.120321,-90.000210
C01169=1913.139200,166.962000,-461.833800,-176.322032,-0.120321,-90.000210
C01170=1911.861000,166.962000,-460.761300,-176.322032,-0.120321,-90.000210
C01171=1908.026200,166.962000,-461.840900,-176.322032,-0.120321,-90.000210
C01172=1906.970100,166.962000,-461.640300,-176.322032,-0.120321,-90.000210
C01173=1902.542000,166.962000,-461.796100,-176.322032,-0.120321,-90.000210
C01174=1901.747200,166.962000,-461.171000,-176.322032,-0.120321,-90.000210
C01175=1897.719000,166.962000,-460.885000,-176.322032,-0.120321,-90.000210
C01176=1896.553500,166.962000,-461.625000,-176.322032,-0.120321,-90.000210
C01177=1894.162500,166.962000,-461.089800,-176.322032,-0.120321,-90.000210
C01178=1891.980800,166.962000,-460.620800,-176.322032,-0.120321,-90.000210
C01179=1890.707200,166.962000,-460.650500,-176.322032,-0.120321,-90.000210
C01180=1887.557200,166.962000,-460.582700,-176.322032,-0.120321,-90.000210
C01181=1886.794600,166.962000,-461.371500,-176.322032,-0.120321,-90.000210
C01182=1885.367300,166.962000,-460.826200,-176.322032,-0.120321,-90.000210
C01183=1881.436400,166.962000,-461.179500,-176.322032,-0.120321,-90.000210
C01184=1880.929900,166.962000,-460.180300,-176.322032,-0.120321,-90.000210
C01185=1876.930000,166.962000,-460.140500,-176.322032,-0.120321,-90.000210
C01186=1876.148900,166.962000,-461.208300,-176.322032,-0.120321,-90.000210
C01187=1872.293300,166.962000,-459.406200,-176.322032,-0.120321,-90.000210
C01188=1871.428200,166.962000,-460.573500,-176.322032,-0.120321,-90.000210
C01189=1867.352500,166.962000,-459.686900,-176.322032,-0.120321,-90.000210
C01190=1866.703100,166.962000,-459.584100,-176.322032,-0.120321,-90.000210
C01191=1864.098700,166.962000,-461.095100,-176.322032,-0.120321,-90.000210
C01192=1862.153100,166.962000,-459.806900,-176.322032,-0.120321,-90.000210
C01193=1861.203700,166.962000,-460.116500,-176.322032,-0.120321,-90.000210
C01194=1857.247700,166.962000,-459.402300,-176.322032,-0.120321,-90.000210
C01195=1856.688700,166.962000,-459.373500,-176.322032,-0.120321,-90.000210
C01196=1852.067900,166.962000,-459.037800,-176.322032,-0.120321,-90.000210
C01197=1851.350900,166.962000,-459.124900,-176.322032,-0.120321,-90.000210
C01198=1847.182700,166.962000,-458.566200,-176.322032,-0.120321,-90.000210
C01199=1846.307300,166.962000,-458.821900,-176.322032,-0.120321,-90.000210
C01200=1842.103200,166.962000,-458.376000,-176.322032,-0.120321,-90.000210
C01201=1841.481400,166.962000,-459.276800,-176.322032,-0.120321,-90.000210
C01202=1837.234200,166.962000,-458.805400,-176.322032,-0.120321,-90.000210
C01203=1836.383200,166.962000,-459.476400,-176.322032,-0.120321,-90.000210
C01204=1832.228000,166.962000,-458.574100,-176.322032,-0.120321,-90.000210
C01205=1830.373100,166.962000,-457.765400,-176.322032,-0.120321,-90.000210
C01206=1826.660200,166.962000,-457.746300,-176.322032,-0.120321,-90.000210
C01207=1825.811300,166.962000,-458.627300,-176.322032,-0.120321,-90.000210
C01208=1821.640300,166.962000,-458.285900,-176.322032,-0.120321,-90.000210
C01209=1820.310800,166.962000,-458.127500,-176.322032,-0.120321,-90.000210
C01210=1817.212000,166.962000,-457.510300,-176.322032,-0.120321,-90.000210
C01211=1816.363800,166.962000,-457.619500,-176.322032,-0.120321,-90.000210
C01212=1812.253400,166.962000,-457.644900,-176.322032,-0.120321,-90.000210
C01213=1810.161500,166.962000,-457.305700,-176.322032,-0.120321,-90.000210
C01214=1807.320000,166.962000,-457.313200,-176.322032,-0.120321,-90.000210
C01215=1805.908300,166.962000,-457.204000,-176.322032,-0.120321,-90.000210
C01216=1802.658500,166.962000,-457.462500,-176.322032,-0.120321,-90.000210
C01217=1801.306500,166.962000,-456.777600,-176.322032,-0.120321,-90.000210
C01218=1797.810900,166.962000,-456.552600,-176.322032,-0.120321,-90.000210
C01219=1796.702900,116.962000,-456.371600,-176.322032,-0.120321,-90.000210
C01220=1797.241700,116.962000,-456.673500,-176.322032,-0.120321,-90.000210
C01221=1800.395900,116.962000,-457.633500,-176.322032,-0.120321,-90.000210
C01222=1801.509300,116.962000,-457.135500,-176.322032,-0.120321,-90.000210
C01223=1806.173400,116.962000,-457.938100,-176.322032,-0.120321,-90.000210
C01224=1807.289000,116.962000,-457.790500,-176.322032,-0.120321,-90.000210
C01225=1811.076300,116.962000,-457.676300,-176.322032,-0.120321,-90.000210
C01226=1812.008900,116.962000,-458.326600,-176.322032,-0.120321,-90.000210
C01227=1814.924100,116.962000,-458.521800,-176.322032,-0.120321,-90.000210
C01228=1816.451800,116.962000,-458.689700,-176.322032,-0.120321,-90.000210
C01229=1820.881300,116.962000,-458.768700,-176.322032,-0.120321,-90.000210
C01230=1821.862600,116.962000,-459.053900,-176.322032,-0.120321,-90.000210
C01231=1825.281700,116.962000,-458.994600,-176.322032,-0.120321,-90.000210
C01232=1826.654000,116.962000,-458.866900,-176.322032,-0.120321,-90.000210
C01233=1831.198900,116.962000,-459.230700,-176.322032,-0.120321,-90.000210
C01234=1831.969400,116.962000,-459.648200,-176.322032,-0.120321,-90.000210
C01235=1834.497600,116.962000,-459.597900,-176.322032,-0.120321,-90.000210
C01236=1836.788700,116.962000,-459.316300,-176.322032,-0.120321,-90.000210
C01237=1841.152400,116.962000,-459.575500,-176.322032,-0.120321,-90.000210
C01238=1842.172600,116.962000,-459.895800,-176.322032,-0.120321,-90.000210
C01239=1845.743900,116.962000,-460.599700,-176.322032,-0.120321,-90.000210
C01240=1847.432600,116.962000,-460.961700,-176.322032,-0.120321,-90.000210
C01241=1847.613500,116.962000,-460.930800,-176.322032,-0.120321,-90.000210
C01242=1851.411300,116.962000,-460.791800,-176.322032,-0.120321,-90.000210
C01243=1852.182400,116.962000,-460.877600,-176.322032,-0.120321,-90.000210
C01244=1853.685900,116.962000,-461.054600,-176.322032,-0.120321,-90.000210
C01245=1856.809900,116.962000,-461.034100,-176.322032,-0.120321,-90.000210
C01246=1857.667700,116.962000,-460.448400,-176.322032,-0.120321,-90.000210
C01247=1861.719700,116.962000,-461.439200,-176.322032,-0.120321,-90.000210
C01248=1862.522500,116.962000,-461.515700,-176.322032,-0.120321,-90.000210
C01249=1863.726100,116.962000,-460.992300,-176.322032,-0.120321,-90.000210
C01250=1866.160400,116.962000,-461.522300,-176.322032,-0.120321,-90.000210
C01251=1868.035200,116.962000,-461.566300,-176.322032,-0.120321,-90.000210
C01252=1871.484400,116.962000,-461.549800,-176.322032,-0.120321,-90.000210
C01253=1872.248500,116.962000,-461.428500,-176.322032,-0.120321,-90.000210
C01254=1876.967500,116.962000,-461.746400,-176.322032,-0.120321,-90.000210
C01255=1877.992200,116.962000,-461.630800,-176.322032,-0.120321,-90.000210
C01256=1881.775700,116.962000,-461.584700,-176.322032,-0.120321,-90.000210
C01257=1882.314000,116.962000,-461.618900,-176.322032,-0.120321,-90.000210
C01258=1886.392900,116.962000,-462.152800,-176.322032,-0.120321,-90.000210
C01259=1887.306100,116.962000,-462.045900,-176.322032,-0.120321,-90.000210
C01260=1891.246500,116.962000,-462.435300,-176.322032,-0.120321,-90.000210
C01261=1892.679600,116.962000,-461.877300,-176.322032,-0.120321,-90.000210
C01262=1896.217500,116.962000,-462.325100,-176.322032,-0.120321,-90.000210
C01263=1898.121300,116.962000,-461.986100,-176.322032,-0.120321,-90.000210
C01264=1901.855900,116.962000,-462.387600,-176.322032,-0.120321,-90.000210
C01265=1902.874800,116.962000,-462.402400,-176.322032,-0.120321,-90.000210
C01266=1907.021400,116.962000,-462.930800,-176.322032,-0.120321,-90.000210
C01267=1907.663600,116.962000,-462.232700,-176.322032,-0.120321,-90.000210
C01268=1910.847000,116.962000,-462.726100,-176.322032,-0.120321,-90.000210
C01269=1911.895000,116.962000,-462.140600,-176.322032,-0.120321,-90.000210
C01270=1916.656200,116.962000,-462.116300,-176.322032,-0.120321,-90.000210
C01271=1918.095800,116.962000,-462.397800,-176.322032,-0.120321,-90.000210
C01272=1921.244100,116.962000,-462.088000,-176.322032,-0.120321,-90.000210
C01273=1921.868500,116.962000,-462.804200,-176.322032,-0.120321,-90.000210
C01274=1926.467200,116.962000,-462.979300,-176.322032,-0.120321,-90.000210
C01275=1927.623500,116.962000,-462.771100,-176.322032,-0.120321,-90.000210
C01276=1931.263700,116.962000,-462.904300,-176.322032,-0.120321,-90.000210
C01277=1932.339400,116.962000,-462.245200,-176.322032,-0.120321,-90.000210
C01278=1936.683600,116.962000,-462.323400,-176.322032,-0.120321,-90.000210
C01279=1938.095900,116.962000,-462.825800,-176.322032,-0.120321,-90.000210
C01280=1941.649200,116.962000,-462.430600,-176.322032,-0.120321,-90.000210
C01281=1942.750600,116.962000,-463.388100,-176.322032,-0.120321,-90.000210
C01282=1946.506000,116.962000,-462.112500,-176.322032,-0.120321,-90.000210
C01283=1947.182400,116.962000,-462.372900,-176.322032,-0.120321,-90.000210
C01284=1951.548700,116.962000,-462.509000,-176.322032,-0.120321,-90.000210
C01285=1952.885600,116.962000,-462.958400,-176.322032,-0.120321,-90.000210
C01286=1957.138700,116.962000,-462.003000,-176.322032,-0.120321,-90.000210
C01287=1958.433700,116.962000,-462.051400,-176.322032,-0.120321,-90.000210
C01288=1961.934400,116.962000,-462.155000,-176.322032,-0.120321,-90.000210
C01289=1962.690700,116.962000,-462.009600,-176.322032,-0.120321,-90.000210
C01290=1966.460500,116.962000,-462.213500,-176.322032,-0.120321,-90.000210
C01291=1968.236400,116.962000,-462.010500,-176.322032,-0.120321,-90.000210
C01292=1971.795000,116.962000,-462.711700,-176.322032,-0.120321,-90.000210
C01293=1972.777700,116.962000,-462.011600,-176.322032,-0.120321,-90.000210
C01294=1976.830800,116.962000,-462.568100,-176.322032,-0.120321,-90.000210
C01295=1977.742900,116.962000,-462.324600,-176.322032,-0.120321,-90.000210
C01296=1982.172700,116.962000,-462.310200,-176.322032,-0.120321,-90.000210
C01297=1982.873800,116.962000,-462.011100,-176.322032,-0.120321,-90.000210
C01298=1986.681900,116.962000,-461.896900,-176.322032,-0.120321,-90.000210
C01299=1987.726300,116.962000,-462.267900,-176.322032,-0.120321,-90.000210
C01300=1992.334400,116.962000,-461.753600,-176.322032,-0.120321,-90.000210
C01301=1993.111800,116.962000,-461.933200,-176.322032,-0.120321,-90.000210
C01302=1996.910100,116.962000,-461.909700,-176.322032,-0.120321,-90.000210
C01303=1997.743200,116.962000,-461.932200,-176.322032,-0.120321,-90.000210
C01304=2001.822700,116.962000,-461.794800,-176.322032,-0.120321,-90.000210
C01305=2002.533400,116.962000,-461.690700,-176.322032,-0.120321,-90.000210
C01306=2006.825000,116.962000,-462.197800,-176.322032,-0.120321,-90.000210
C01307=2009.014700,116.962000,-462.283400,-176.322032,-0.120321,-90.000210
C01308=2011.856400,116.962000,-461.956700,-176.322032,-0.120321,-90.000210
C01309=2012.956000,116.962000,-461.497900,-176.322032,-0.120321,-90.000210
C01310=2016.564200,116.962000,-462.058000,-176.322032,-0.120321,-90.000210
C01311=2017.673700,116.962000,-461.608100,-176.322032,-0.120321,-90.000210
C01312=2021.695200,116.962000,-461.898800,-176.322032,-0.120321,-90.000210
C01313=2022.942700,116.962000,-462.144000,-176.322032,-0.120321,-90.000210
C01314=2026.672400,116.962000,-461.435000,-176.322032,-0.120321,-90.000210
C01315=2027.498500,116.962000,-461.854800,-176.322032,-0.120321,-90.000210
C01316=2031.461200,116.962000,-461.818100,-176.322032,-0.120321,-90.000210
C01317=2033.422600,116.962000,-461.251100,-176.322032,-0.120321,-90.000210
